      A     M      3.3;
      =     L      0.0;
      A(    ;
      A(    ;
      A     L      0.0;
      AN    M   2002.7;
      JNB   _001;
      L     0;
      T     MW  2150;
      SET   ;
      SAVE  ;
      CLR   ;
_001: A     BR;
      )     ;
      JNB   _002;
      L     0;
      T     MW  2152;
      SET   ;
      SAVE  ;
      CLR   ;
_002: A     BR;
      )     ;
      JNB   _003;
      L     0;
      T     MB  2154;
_003: NOP   0;
      A(    ;
      A(    ;
      A     L      0.0;
      AN    M   2002.5;
      JNB   _004;
      L     0;
      T     MW  2250;
      SET   ;
      SAVE  ;
      CLR   ;
_004: A     BR;
      )     ;
      JNB   _005;
      L     0;
      T     MW  2252;
      SET   ;
      SAVE  ;
      CLR   ;
_005: A     BR;
      )     ;
      JNB   _006;
      L     0;
      T     MB  2254;
_006: NOP   0;
NETWORK
TITLE =
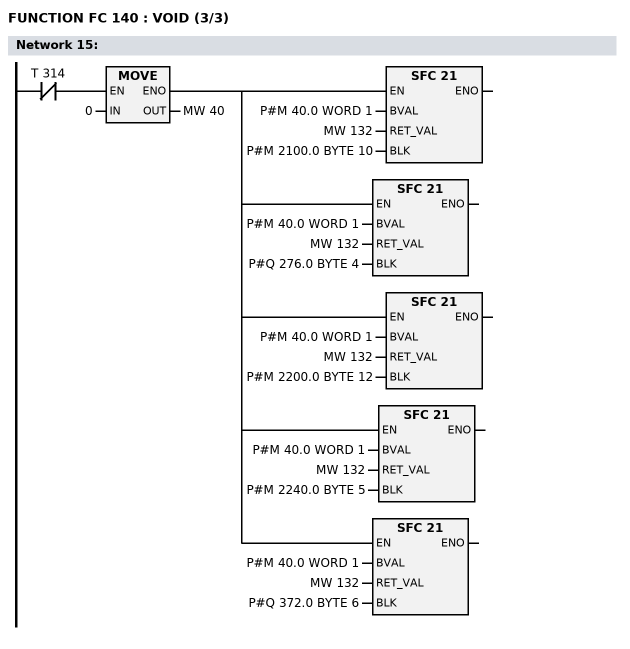

      AN    T    314;
      JNB   _007;
      L     0;
      T     MW    40;
      SET   ;
      SAVE  ;
      CLR   ;
_007: A     BR;
      =     L      0.0;
      A     L      0.0;
      JNB   _008;
      CALL SFC   21 (
           BVAL                     := P#M 40.0 WORD 1,
           RET_VAL                  := MW   132,
           BLK                      := P#M 2100.0 BYTE 10);
_008: NOP   0;
      A     L      0.0;
      JNB   _009;
      CALL SFC   21 (
           BVAL                     := P#M 40.0 WORD 1,
           RET_VAL                  := MW   132,
           BLK                      := P#Q 276.0 BYTE 4);
_009: NOP   0;
      A     L      0.0;
      JNB   _00a;
      CALL SFC   21 (
           BVAL                     := P#M 40.0 WORD 1,
           RET_VAL                  := MW   132,
           BLK                      := P#M 2200.0 BYTE 12);
_00a: NOP   0;
      A     L      0.0;
      JNB   _00b;
      CALL SFC   21 (
           BVAL                     := P#M 40.0 WORD 1,
           RET_VAL                  := MW   132,
           BLK                      := P#M 2240.0 BYTE 5);
_00b: NOP   0;
      A     L      0.0;
      JNB   _00c;
      CALL SFC   21 (
           BVAL                     := P#M 40.0 WORD 1,
           RET_VAL                  := MW   132,
           BLK                      := P#Q 372.0 BYTE 6);
_00c: NOP   0;
END_FUNCTION

FUNCTION_BLOCK FB 141
TITLE =
VERSION : 0.1


VAR
  S704_HOOK_PIN : FB 424;
  S704_DAECHA_LOCK : FB 424;
  S704_ELE : FB 424;
  S704_AIR_ELE : FB 424;
  S704_FF_OUT_CLAMP : FB 424;
END_VAR
BEGIN
NETWORK
TITLE =
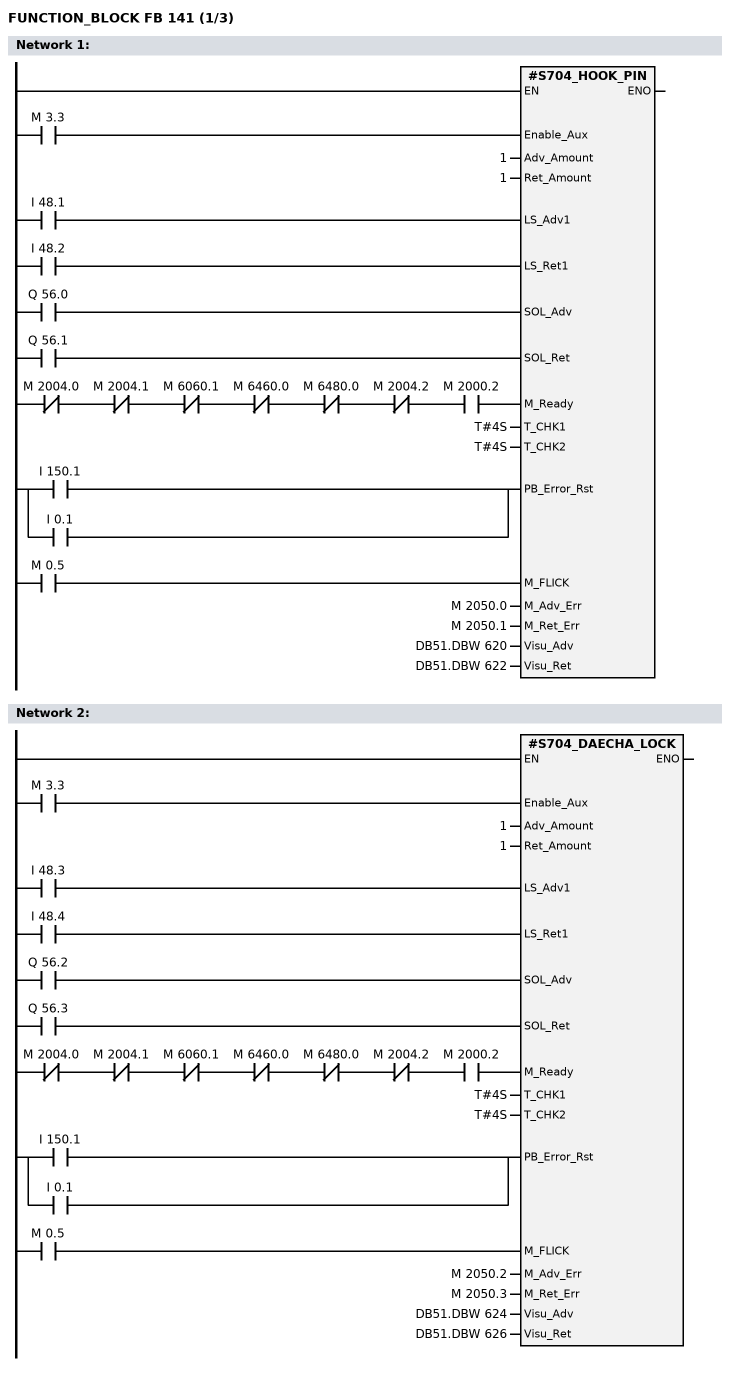

      A     M      3.3;
      =     L      0.0;
      BLD   103;
      A     I     48.1;
      =     L      0.1;
      BLD   103;
      A     I     48.2;
      =     L      0.2;
      BLD   103;
      A     Q     56.0;
      =     L      1.1;
      BLD   103;
      A     Q     56.1;
      =     L      1.2;
      BLD   103;
      AN    M   2004.0;
      AN    M   2004.1;
      AN    M   6060.1;
      AN    M   6460.0;
      AN    M   6480.0;
      AN    M   2004.2;
      A     M   2000.2;
      =     L      1.3;
      BLD   103;
      A(    ;
      O     I    150.1;
      O     I      0.1;
      )     ;
      =     L      1.5;
      BLD   103;
      A     M      0.5;
      =     L      1.6;
      BLD   103;
      CALL #S704_HOOK_PIN (
           Enable_Aux               := L      0.0,
           Adv_Amount               := 1,
           Ret_Amount               := 1,
           LS_Adv1                  := L      0.1,
           LS_Ret1                  := L      0.2,
           SOL_Adv                  := L      1.1,
           SOL_Ret                  := L      1.2,
           M_Ready                  := L      1.3,
           T_CHK1                   := T#4S,
           T_CHK2                   := T#4S,
           PB_Error_Rst             := L      1.5,
           M_FLICK                  := L      1.6,
           M_Adv_Err                := M   2050.0,
           M_Ret_Err                := M   2050.1,
           Visu_Adv                 := DB51.DBW  620,
           Visu_Ret                 := DB51.DBW  622);
      NOP   0;
NETWORK
TITLE =

      A     M      3.3;
      =     L      0.0;
      BLD   103;
      A     I     48.3;
      =     L      0.1;
      BLD   103;
      A     I     48.4;
      =     L      0.2;
      BLD   103;
      A     Q     56.2;
      =     L      1.1;
      BLD   103;
      A     Q     56.3;
      =     L      1.2;
      BLD   103;
      AN    M   2004.0;
      AN    M   2004.1;
      AN    M   6060.1;
      AN    M   6460.0;
      AN    M   6480.0;
      AN    M   2004.2;
      A     M   2000.2;
      =     L      1.3;
      BLD   103;
      A(    ;
      O     I    150.1;
      O     I      0.1;
      )     ;
      =     L      1.5;
      BLD   103;
      A     M      0.5;
      =     L      1.6;
      BLD   103;
      CALL #S704_DAECHA_LOCK (
           Enable_Aux               := L      0.0,
           Adv_Amount               := 1,
           Ret_Amount               := 1,
           LS_Adv1                  := L      0.1,
           LS_Ret1                  := L      0.2,
           SOL_Adv                  := L      1.1,
           SOL_Ret                  := L      1.2,
           M_Ready                  := L      1.3,
           T_CHK1                   := T#4S,
           T_CHK2                   := T#4S,
           PB_Error_Rst             := L      1.5,
           M_FLICK                  := L      1.6,
           M_Adv_Err                := M   2050.2,
           M_Ret_Err                := M   2050.3,
           Visu_Adv                 := DB51.DBW  624,
           Visu_Ret                 := DB51.DBW  626);
      NOP   0;
NETWORK
TITLE =
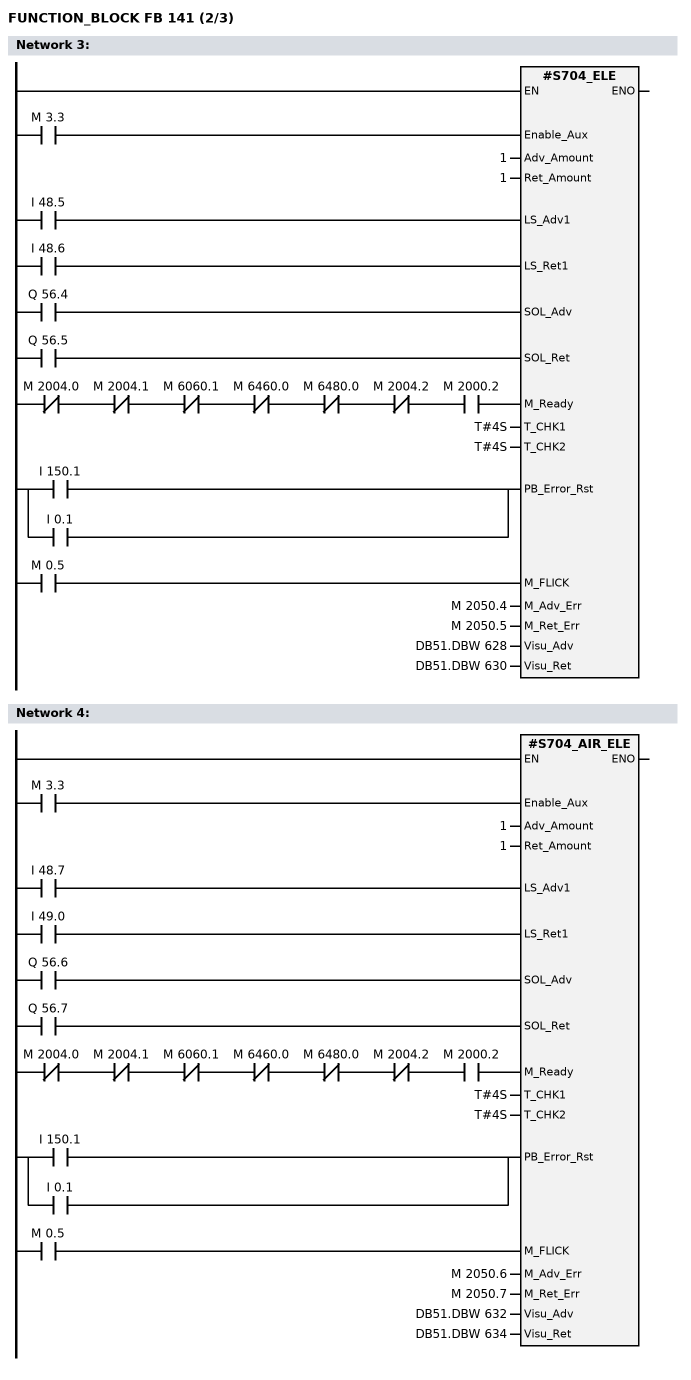

      A     M      3.3;
      =     L      0.0;
      BLD   103;
      A     I     48.5;
      =     L      0.1;
      BLD   103;
      A     I     48.6;
      =     L      0.2;
      BLD   103;
      A     Q     56.4;
      =     L      1.1;
      BLD   103;
      A     Q     56.5;
      =     L      1.2;
      BLD   103;
      AN    M   2004.0;
      AN    M   2004.1;
      AN    M   6060.1;
      AN    M   6460.0;
      AN    M   6480.0;
      AN    M   2004.2;
      A     M   2000.2;
      =     L      1.3;
      BLD   103;
      A(    ;
      O     I    150.1;
      O     I      0.1;
      )     ;
      =     L      1.5;
      BLD   103;
      A     M      0.5;
      =     L      1.6;
      BLD   103;
      CALL #S704_ELE (
           Enable_Aux               := L      0.0,
           Adv_Amount               := 1,
           Ret_Amount               := 1,
           LS_Adv1                  := L      0.1,
           LS_Ret1                  := L      0.2,
           SOL_Adv                  := L      1.1,
           SOL_Ret                  := L      1.2,
           M_Ready                  := L      1.3,
           T_CHK1                   := T#4S,
           T_CHK2                   := T#4S,
           PB_Error_Rst             := L      1.5,
           M_FLICK                  := L      1.6,
           M_Adv_Err                := M   2050.4,
           M_Ret_Err                := M   2050.5,
           Visu_Adv                 := DB51.DBW  628,
           Visu_Ret                 := DB51.DBW  630);
      NOP   0;
NETWORK
TITLE =

      A     M      3.3;
      =     L      0.0;
      BLD   103;
      A     I     48.7;
      =     L      0.1;
      BLD   103;
      A     I     49.0;
      =     L      0.2;
      BLD   103;
      A     Q     56.6;
      =     L      1.1;
      BLD   103;
      A     Q     56.7;
      =     L      1.2;
      BLD   103;
      AN    M   2004.0;
      AN    M   2004.1;
      AN    M   6060.1;
      AN    M   6460.0;
      AN    M   6480.0;
      AN    M   2004.2;
      A     M   2000.2;
      =     L      1.3;
      BLD   103;
      A(    ;
      O     I    150.1;
      O     I      0.1;
      )     ;
      =     L      1.5;
      BLD   103;
      A     M      0.5;
      =     L      1.6;
      BLD   103;
      CALL #S704_AIR_ELE (
           Enable_Aux               := L      0.0,
           Adv_Amount               := 1,
           Ret_Amount               := 1,
           LS_Adv1                  := L      0.1,
           LS_Ret1                  := L      0.2,
           SOL_Adv                  := L      1.1,
           SOL_Ret                  := L      1.2,
           M_Ready                  := L      1.3,
           T_CHK1                   := T#4S,
           T_CHK2                   := T#4S,
           PB_Error_Rst             := L      1.5,
           M_FLICK                  := L      1.6,
           M_Adv_Err                := M   2050.6,
           M_Ret_Err                := M   2050.7,
           Visu_Adv                 := DB51.DBW  632,
           Visu_Ret                 := DB51.DBW  634);
      NOP   0;
NETWORK
TITLE =
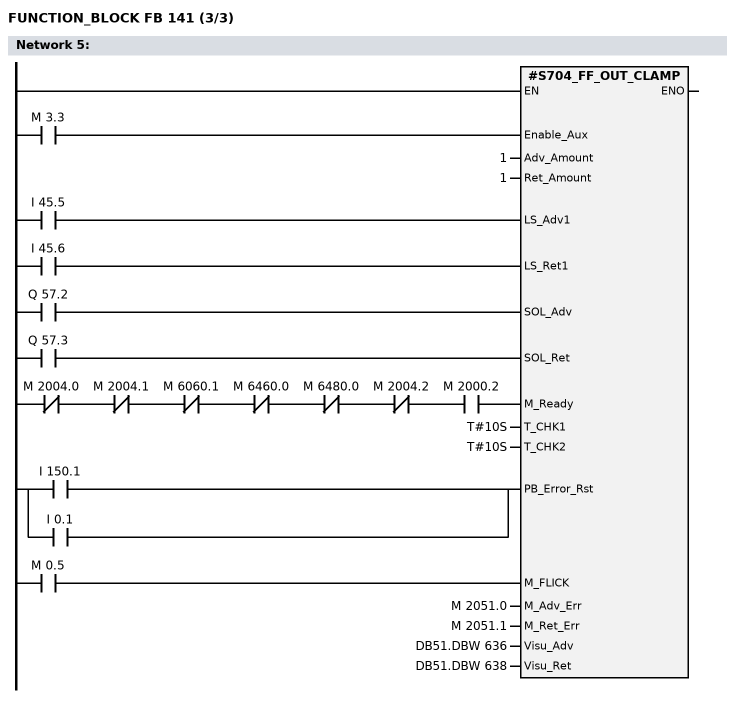

      A     M      3.3;
      =     L      0.0;
      BLD   103;
      A     I     45.5;
      =     L      0.1;
      BLD   103;
      A     I     45.6;
      =     L      0.2;
      BLD   103;
      A     Q     57.2;
      =     L      1.1;
      BLD   103;
      A     Q     57.3;
      =     L      1.2;
      BLD   103;
      AN    M   2004.0;
      AN    M   2004.1;
      AN    M   6060.1;
      AN    M   6460.0;
      AN    M   6480.0;
      AN    M   2004.2;
      A     M   2000.2;
      =     L      1.3;
      BLD   103;
      A(    ;
      O     I    150.1;
      O     I      0.1;
      )     ;
      =     L      1.5;
      BLD   103;
      A     M      0.5;
      =     L      1.6;
      BLD   103;
      CALL #S704_FF_OUT_CLAMP (
           Enable_Aux               := L      0.0,
           Adv_Amount               := 1,
           Ret_Amount               := 1,
           LS_Adv1                  := L      0.1,
           LS_Ret1                  := L      0.2,
           SOL_Adv                  := L      1.1,
           SOL_Ret                  := L      1.2,
           M_Ready                  := L      1.3,
           T_CHK1                   := T#10S,
           T_CHK2                   := T#10S,
           PB_Error_Rst             := L      1.5,
           M_FLICK                  := L      1.6,
           M_Adv_Err                := M   2051.0,
           M_Ret_Err                := M   2051.1,
           Visu_Adv                 := DB51.DBW  636,
           Visu_Ret                 := DB51.DBW  638);
      NOP   0;
END_FUNCTION_BLOCK

DATA_BLOCK DB 141
TITLE =
VERSION : 0.0

 FB 141
BEGIN
   S704_HOOK_PIN.Enable_Aux := FALSE;
   S704_HOOK_PIN.Adv_Amount := 0;
   S704_HOOK_PIN.Ret_Amount := 0;
   S704_HOOK_PIN.LS_Adv1 := FALSE;
   S704_HOOK_PIN.LS_Ret1 := FALSE;
   S704_HOOK_PIN.LS_Adv2 := FALSE;
   S704_HOOK_PIN.LS_Ret2 := FALSE;
   S704_HOOK_PIN.LS_Adv3 := FALSE;
   S704_HOOK_PIN.LS_Ret3 := FALSE;
   S704_HOOK_PIN.LS_Adv4 := FALSE;
   S704_HOOK_PIN.LS_Ret4 := FALSE;
   S704_HOOK_PIN.SOL_Adv := FALSE;
   S704_HOOK_PIN.SOL_Ret := FALSE;
   S704_HOOK_PIN.M_Ready := FALSE;
   S704_HOOK_PIN.T_CHK1 := T#0MS;
   S704_HOOK_PIN.T_CHK2 := T#0MS;
   S704_HOOK_PIN.PB_Lamp_CHK := FALSE;
   S704_HOOK_PIN.PB_Error_Rst := FALSE;
   S704_HOOK_PIN.M_FLICK := FALSE;
   S704_HOOK_PIN.M_Adv_Err := FALSE;
   S704_HOOK_PIN.M_Ret_Err := FALSE;
   S704_HOOK_PIN.LP_Adv := FALSE;
   S704_HOOK_PIN.LP_Ret := FALSE;
   S704_HOOK_PIN.Visu_Adv := W#16#0;
   S704_HOOK_PIN.Visu_Ret := W#16#0;
   S704_HOOK_PIN.Error_T1.IN := FALSE;
   S704_HOOK_PIN.Error_T1.PT := T#0MS;
   S704_HOOK_PIN.Error_T1.Q := FALSE;
   S704_HOOK_PIN.Error_T1.ET := T#0MS;
   S704_HOOK_PIN.Error_T1.STATE := B#16#0;
   S704_HOOK_PIN.Error_T1.STIME := T#0MS;
   S704_HOOK_PIN.Error_T1.ATIME := T#0MS;
   S704_HOOK_PIN.Error_T2.IN := FALSE;
   S704_HOOK_PIN.Error_T2.PT := T#0MS;
   S704_HOOK_PIN.Error_T2.Q := FALSE;
   S704_HOOK_PIN.Error_T2.ET := T#0MS;
   S704_HOOK_PIN.Error_T2.STATE := B#16#0;
   S704_HOOK_PIN.Error_T2.STIME := T#0MS;
   S704_HOOK_PIN.Error_T2.ATIME := T#0MS;
   S704_HOOK_PIN.CHK_Aux1 := FALSE;
   S704_HOOK_PIN.CHK_Aux2 := FALSE;
   S704_HOOK_PIN.Error_T1_DN := FALSE;
   S704_HOOK_PIN.Error_T2_DN := FALSE;
   S704_HOOK_PIN.Adv_Memo := FALSE;
   S704_HOOK_PIN.Visu_Adv_Arr[0] := FALSE;
   S704_HOOK_PIN.Visu_Adv_Arr[1] := FALSE;
   S704_HOOK_PIN.Visu_Adv_Arr[2] := FALSE;
   S704_HOOK_PIN.Visu_Adv_Arr[3] := FALSE;
   S704_HOOK_PIN.Visu_Adv_Arr[4] := FALSE;
   S704_HOOK_PIN.Visu_Adv_Arr[5] := FALSE;
   S704_HOOK_PIN.Visu_Adv_Arr[6] := FALSE;
   S704_HOOK_PIN.Visu_Adv_Arr[7] := FALSE;
   S704_HOOK_PIN.Visu_Adv_Arr[8] := FALSE;
   S704_HOOK_PIN.Visu_Adv_Arr[9] := FALSE;
   S704_HOOK_PIN.Visu_Adv_Arr[10] := FALSE;
   S704_HOOK_PIN.Visu_Adv_Arr[11] := FALSE;
   S704_HOOK_PIN.Visu_Adv_Arr[12] := FALSE;
   S704_HOOK_PIN.Visu_Adv_Arr[13] := FALSE;
   S704_HOOK_PIN.Visu_Adv_Arr[14] := FALSE;
   S704_HOOK_PIN.Visu_Adv_Arr[15] := FALSE;
   S704_HOOK_PIN.Visu_Ret_Arr[0] := FALSE;
   S704_HOOK_PIN.Visu_Ret_Arr[1] := FALSE;
   S704_HOOK_PIN.Visu_Ret_Arr[2] := FALSE;
   S704_HOOK_PIN.Visu_Ret_Arr[3] := FALSE;
   S704_HOOK_PIN.Visu_Ret_Arr[4] := FALSE;
   S704_HOOK_PIN.Visu_Ret_Arr[5] := FALSE;
   S704_HOOK_PIN.Visu_Ret_Arr[6] := FALSE;
   S704_HOOK_PIN.Visu_Ret_Arr[7] := FALSE;
   S704_HOOK_PIN.Visu_Ret_Arr[8] := FALSE;
   S704_HOOK_PIN.Visu_Ret_Arr[9] := FALSE;
   S704_HOOK_PIN.Visu_Ret_Arr[10] := FALSE;
   S704_HOOK_PIN.Visu_Ret_Arr[11] := FALSE;
   S704_HOOK_PIN.Visu_Ret_Arr[12] := FALSE;
   S704_HOOK_PIN.Visu_Ret_Arr[13] := FALSE;
   S704_HOOK_PIN.Visu_Ret_Arr[14] := FALSE;
   S704_HOOK_PIN.Visu_Ret_Arr[15] := FALSE;
   S704_HOOK_PIN.BLK_Move_Ret := 0;
   S704_HOOK_PIN.Enable := FALSE;
   S704_HOOK_PIN.Adv_End := FALSE;
   S704_HOOK_PIN.Ret_End := FALSE;
   S704_DAECHA_LOCK.Enable_Aux := FALSE;
   S704_DAECHA_LOCK.Adv_Amount := 0;
   S704_DAECHA_LOCK.Ret_Amount := 0;
   S704_DAECHA_LOCK.LS_Adv1 := FALSE;
   S704_DAECHA_LOCK.LS_Ret1 := FALSE;
   S704_DAECHA_LOCK.LS_Adv2 := FALSE;
   S704_DAECHA_LOCK.LS_Ret2 := FALSE;
   S704_DAECHA_LOCK.LS_Adv3 := FALSE;
   S704_DAECHA_LOCK.LS_Ret3 := FALSE;
   S704_DAECHA_LOCK.LS_Adv4 := FALSE;
   S704_DAECHA_LOCK.LS_Ret4 := FALSE;
   S704_DAECHA_LOCK.SOL_Adv := FALSE;
   S704_DAECHA_LOCK.SOL_Ret := FALSE;
   S704_DAECHA_LOCK.M_Ready := FALSE;
   S704_DAECHA_LOCK.T_CHK1 := T#0MS;
   S704_DAECHA_LOCK.T_CHK2 := T#0MS;
   S704_DAECHA_LOCK.PB_Lamp_CHK := FALSE;
   S704_DAECHA_LOCK.PB_Error_Rst := FALSE;
   S704_DAECHA_LOCK.M_FLICK := FALSE;
   S704_DAECHA_LOCK.M_Adv_Err := FALSE;
   S704_DAECHA_LOCK.M_Ret_Err := FALSE;
   S704_DAECHA_LOCK.LP_Adv := FALSE;
   S704_DAECHA_LOCK.LP_Ret := FALSE;
   S704_DAECHA_LOCK.Visu_Adv := W#16#0;
   S704_DAECHA_LOCK.Visu_Ret := W#16#0;
   S704_DAECHA_LOCK.Error_T1.IN := FALSE;
   S704_DAECHA_LOCK.Error_T1.PT := T#0MS;
   S704_DAECHA_LOCK.Error_T1.Q := FALSE;
   S704_DAECHA_LOCK.Error_T1.ET := T#0MS;
   S704_DAECHA_LOCK.Error_T1.STATE := B#16#0;
   S704_DAECHA_LOCK.Error_T1.STIME := T#0MS;
   S704_DAECHA_LOCK.Error_T1.ATIME := T#0MS;
   S704_DAECHA_LOCK.Error_T2.IN := FALSE;
   S704_DAECHA_LOCK.Error_T2.PT := T#0MS;
   S704_DAECHA_LOCK.Error_T2.Q := FALSE;
   S704_DAECHA_LOCK.Error_T2.ET := T#0MS;
   S704_DAECHA_LOCK.Error_T2.STATE := B#16#0;
   S704_DAECHA_LOCK.Error_T2.STIME := T#0MS;
   S704_DAECHA_LOCK.Error_T2.ATIME := T#0MS;
   S704_DAECHA_LOCK.CHK_Aux1 := FALSE;
   S704_DAECHA_LOCK.CHK_Aux2 := FALSE;
   S704_DAECHA_LOCK.Error_T1_DN := FALSE;
   S704_DAECHA_LOCK.Error_T2_DN := FALSE;
   S704_DAECHA_LOCK.Adv_Memo := FALSE;
   S704_DAECHA_LOCK.Visu_Adv_Arr[0] := FALSE;
   S704_DAECHA_LOCK.Visu_Adv_Arr[1] := FALSE;
   S704_DAECHA_LOCK.Visu_Adv_Arr[2] := FALSE;
   S704_DAECHA_LOCK.Visu_Adv_Arr[3] := FALSE;
   S704_DAECHA_LOCK.Visu_Adv_Arr[4] := FALSE;
   S704_DAECHA_LOCK.Visu_Adv_Arr[5] := FALSE;
   S704_DAECHA_LOCK.Visu_Adv_Arr[6] := FALSE;
   S704_DAECHA_LOCK.Visu_Adv_Arr[7] := FALSE;
   S704_DAECHA_LOCK.Visu_Adv_Arr[8] := FALSE;
   S704_DAECHA_LOCK.Visu_Adv_Arr[9] := FALSE;
   S704_DAECHA_LOCK.Visu_Adv_Arr[10] := FALSE;
   S704_DAECHA_LOCK.Visu_Adv_Arr[11] := FALSE;
   S704_DAECHA_LOCK.Visu_Adv_Arr[12] := FALSE;
   S704_DAECHA_LOCK.Visu_Adv_Arr[13] := FALSE;
   S704_DAECHA_LOCK.Visu_Adv_Arr[14] := FALSE;
   S704_DAECHA_LOCK.Visu_Adv_Arr[15] := FALSE;
   S704_DAECHA_LOCK.Visu_Ret_Arr[0] := FALSE;
   S704_DAECHA_LOCK.Visu_Ret_Arr[1] := FALSE;
   S704_DAECHA_LOCK.Visu_Ret_Arr[2] := FALSE;
   S704_DAECHA_LOCK.Visu_Ret_Arr[3] := FALSE;
   S704_DAECHA_LOCK.Visu_Ret_Arr[4] := FALSE;
   S704_DAECHA_LOCK.Visu_Ret_Arr[5] := FALSE;
   S704_DAECHA_LOCK.Visu_Ret_Arr[6] := FALSE;
   S704_DAECHA_LOCK.Visu_Ret_Arr[7] := FALSE;
   S704_DAECHA_LOCK.Visu_Ret_Arr[8] := FALSE;
   S704_DAECHA_LOCK.Visu_Ret_Arr[9] := FALSE;
   S704_DAECHA_LOCK.Visu_Ret_Arr[10] := FALSE;
   S704_DAECHA_LOCK.Visu_Ret_Arr[11] := FALSE;
   S704_DAECHA_LOCK.Visu_Ret_Arr[12] := FALSE;
   S704_DAECHA_LOCK.Visu_Ret_Arr[13] := FALSE;
   S704_DAECHA_LOCK.Visu_Ret_Arr[14] := FALSE;
   S704_DAECHA_LOCK.Visu_Ret_Arr[15] := FALSE;
   S704_DAECHA_LOCK.BLK_Move_Ret := 0;
   S704_DAECHA_LOCK.Enable := FALSE;
   S704_DAECHA_LOCK.Adv_End := FALSE;
   S704_DAECHA_LOCK.Ret_End := FALSE;
   S704_ELE.Enable_Aux := FALSE;
   S704_ELE.Adv_Amount := 0;
   S704_ELE.Ret_Amount := 0;
   S704_ELE.LS_Adv1 := FALSE;
   S704_ELE.LS_Ret1 := FALSE;
   S704_ELE.LS_Adv2 := FALSE;
   S704_ELE.LS_Ret2 := FALSE;
   S704_ELE.LS_Adv3 := FALSE;
   S704_ELE.LS_Ret3 := FALSE;
   S704_ELE.LS_Adv4 := FALSE;
   S704_ELE.LS_Ret4 := FALSE;
   S704_ELE.SOL_Adv := FALSE;
   S704_ELE.SOL_Ret := FALSE;
   S704_ELE.M_Ready := FALSE;
   S704_ELE.T_CHK1 := T#0MS;
   S704_ELE.T_CHK2 := T#0MS;
   S704_ELE.PB_Lamp_CHK := FALSE;
   S704_ELE.PB_Error_Rst := FALSE;
   S704_ELE.M_FLICK := FALSE;
   S704_ELE.M_Adv_Err := FALSE;
   S704_ELE.M_Ret_Err := FALSE;
   S704_ELE.LP_Adv := FALSE;
   S704_ELE.LP_Ret := FALSE;
   S704_ELE.Visu_Adv := W#16#0;
   S704_ELE.Visu_Ret := W#16#0;
   S704_ELE.Error_T1.IN := FALSE;
   S704_ELE.Error_T1.PT := T#0MS;
   S704_ELE.Error_T1.Q := FALSE;
   S704_ELE.Error_T1.ET := T#0MS;
   S704_ELE.Error_T1.STATE := B#16#0;
   S704_ELE.Error_T1.STIME := T#0MS;
   S704_ELE.Error_T1.ATIME := T#0MS;
   S704_ELE.Error_T2.IN := FALSE;
   S704_ELE.Error_T2.PT := T#0MS;
   S704_ELE.Error_T2.Q := FALSE;
   S704_ELE.Error_T2.ET := T#0MS;
   S704_ELE.Error_T2.STATE := B#16#0;
   S704_ELE.Error_T2.STIME := T#0MS;
   S704_ELE.Error_T2.ATIME := T#0MS;
   S704_ELE.CHK_Aux1 := FALSE;
   S704_ELE.CHK_Aux2 := FALSE;
   S704_ELE.Error_T1_DN := FALSE;
   S704_ELE.Error_T2_DN := FALSE;
   S704_ELE.Adv_Memo := FALSE;
   S704_ELE.Visu_Adv_Arr[0] := FALSE;
   S704_ELE.Visu_Adv_Arr[1] := FALSE;
   S704_ELE.Visu_Adv_Arr[2] := FALSE;
   S704_ELE.Visu_Adv_Arr[3] := FALSE;
   S704_ELE.Visu_Adv_Arr[4] := FALSE;
   S704_ELE.Visu_Adv_Arr[5] := FALSE;
   S704_ELE.Visu_Adv_Arr[6] := FALSE;
   S704_ELE.Visu_Adv_Arr[7] := FALSE;
   S704_ELE.Visu_Adv_Arr[8] := FALSE;
   S704_ELE.Visu_Adv_Arr[9] := FALSE;
   S704_ELE.Visu_Adv_Arr[10] := FALSE;
   S704_ELE.Visu_Adv_Arr[11] := FALSE;
   S704_ELE.Visu_Adv_Arr[12] := FALSE;
   S704_ELE.Visu_Adv_Arr[13] := FALSE;
   S704_ELE.Visu_Adv_Arr[14] := FALSE;
   S704_ELE.Visu_Adv_Arr[15] := FALSE;
   S704_ELE.Visu_Ret_Arr[0] := FALSE;
   S704_ELE.Visu_Ret_Arr[1] := FALSE;
   S704_ELE.Visu_Ret_Arr[2] := FALSE;
   S704_ELE.Visu_Ret_Arr[3] := FALSE;
   S704_ELE.Visu_Ret_Arr[4] := FALSE;
   S704_ELE.Visu_Ret_Arr[5] := FALSE;
   S704_ELE.Visu_Ret_Arr[6] := FALSE;
   S704_ELE.Visu_Ret_Arr[7] := FALSE;
   S704_ELE.Visu_Ret_Arr[8] := FALSE;
   S704_ELE.Visu_Ret_Arr[9] := FALSE;
   S704_ELE.Visu_Ret_Arr[10] := FALSE;
   S704_ELE.Visu_Ret_Arr[11] := FALSE;
   S704_ELE.Visu_Ret_Arr[12] := FALSE;
   S704_ELE.Visu_Ret_Arr[13] := FALSE;
   S704_ELE.Visu_Ret_Arr[14] := FALSE;
   S704_ELE.Visu_Ret_Arr[15] := FALSE;
   S704_ELE.BLK_Move_Ret := 0;
   S704_ELE.Enable := FALSE;
   S704_ELE.Adv_End := FALSE;
   S704_ELE.Ret_End := FALSE;
   S704_AIR_ELE.Enable_Aux := FALSE;
   S704_AIR_ELE.Adv_Amount := 0;
   S704_AIR_ELE.Ret_Amount := 0;
   S704_AIR_ELE.LS_Adv1 := FALSE;
   S704_AIR_ELE.LS_Ret1 := FALSE;
   S704_AIR_ELE.LS_Adv2 := FALSE;
   S704_AIR_ELE.LS_Ret2 := FALSE;
   S704_AIR_ELE.LS_Adv3 := FALSE;
   S704_AIR_ELE.LS_Ret3 := FALSE;
   S704_AIR_ELE.LS_Adv4 := FALSE;
   S704_AIR_ELE.LS_Ret4 := FALSE;
   S704_AIR_ELE.SOL_Adv := FALSE;
   S704_AIR_ELE.SOL_Ret := FALSE;
   S704_AIR_ELE.M_Ready := FALSE;
   S704_AIR_ELE.T_CHK1 := T#0MS;
   S704_AIR_ELE.T_CHK2 := T#0MS;
   S704_AIR_ELE.PB_Lamp_CHK := FALSE;
   S704_AIR_ELE.PB_Error_Rst := FALSE;
   S704_AIR_ELE.M_FLICK := FALSE;
   S704_AIR_ELE.M_Adv_Err := FALSE;
   S704_AIR_ELE.M_Ret_Err := FALSE;
   S704_AIR_ELE.LP_Adv := FALSE;
   S704_AIR_ELE.LP_Ret := FALSE;
   S704_AIR_ELE.Visu_Adv := W#16#0;
   S704_AIR_ELE.Visu_Ret := W#16#0;
   S704_AIR_ELE.Error_T1.IN := FALSE;
   S704_AIR_ELE.Error_T1.PT := T#0MS;
   S704_AIR_ELE.Error_T1.Q := FALSE;
   S704_AIR_ELE.Error_T1.ET := T#0MS;
   S704_AIR_ELE.Error_T1.STATE := B#16#0;
   S704_AIR_ELE.Error_T1.STIME := T#0MS;
   S704_AIR_ELE.Error_T1.ATIME := T#0MS;
   S704_AIR_ELE.Error_T2.IN := FALSE;
   S704_AIR_ELE.Error_T2.PT := T#0MS;
   S704_AIR_ELE.Error_T2.Q := FALSE;
   S704_AIR_ELE.Error_T2.ET := T#0MS;
   S704_AIR_ELE.Error_T2.STATE := B#16#0;
   S704_AIR_ELE.Error_T2.STIME := T#0MS;
   S704_AIR_ELE.Error_T2.ATIME := T#0MS;
   S704_AIR_ELE.CHK_Aux1 := FALSE;
   S704_AIR_ELE.CHK_Aux2 := FALSE;
   S704_AIR_ELE.Error_T1_DN := FALSE;
   S704_AIR_ELE.Error_T2_DN := FALSE;
   S704_AIR_ELE.Adv_Memo := FALSE;
   S704_AIR_ELE.Visu_Adv_Arr[0] := FALSE;
   S704_AIR_ELE.Visu_Adv_Arr[1] := FALSE;
   S704_AIR_ELE.Visu_Adv_Arr[2] := FALSE;
   S704_AIR_ELE.Visu_Adv_Arr[3] := FALSE;
   S704_AIR_ELE.Visu_Adv_Arr[4] := FALSE;
   S704_AIR_ELE.Visu_Adv_Arr[5] := FALSE;
   S704_AIR_ELE.Visu_Adv_Arr[6] := FALSE;
   S704_AIR_ELE.Visu_Adv_Arr[7] := FALSE;
   S704_AIR_ELE.Visu_Adv_Arr[8] := FALSE;
   S704_AIR_ELE.Visu_Adv_Arr[9] := FALSE;
   S704_AIR_ELE.Visu_Adv_Arr[10] := FALSE;
   S704_AIR_ELE.Visu_Adv_Arr[11] := FALSE;
   S704_AIR_ELE.Visu_Adv_Arr[12] := FALSE;
   S704_AIR_ELE.Visu_Adv_Arr[13] := FALSE;
   S704_AIR_ELE.Visu_Adv_Arr[14] := FALSE;
   S704_AIR_ELE.Visu_Adv_Arr[15] := FALSE;
   S704_AIR_ELE.Visu_Ret_Arr[0] := FALSE;
   S704_AIR_ELE.Visu_Ret_Arr[1] := FALSE;
   S704_AIR_ELE.Visu_Ret_Arr[2] := FALSE;
   S704_AIR_ELE.Visu_Ret_Arr[3] := FALSE;
   S704_AIR_ELE.Visu_Ret_Arr[4] := FALSE;
   S704_AIR_ELE.Visu_Ret_Arr[5] := FALSE;
   S704_AIR_ELE.Visu_Ret_Arr[6] := FALSE;
   S704_AIR_ELE.Visu_Ret_Arr[7] := FALSE;
   S704_AIR_ELE.Visu_Ret_Arr[8] := FALSE;
   S704_AIR_ELE.Visu_Ret_Arr[9] := FALSE;
   S704_AIR_ELE.Visu_Ret_Arr[10] := FALSE;
   S704_AIR_ELE.Visu_Ret_Arr[11] := FALSE;
   S704_AIR_ELE.Visu_Ret_Arr[12] := FALSE;
   S704_AIR_ELE.Visu_Ret_Arr[13] := FALSE;
   S704_AIR_ELE.Visu_Ret_Arr[14] := FALSE;
   S704_AIR_ELE.Visu_Ret_Arr[15] := FALSE;
   S704_AIR_ELE.BLK_Move_Ret := 0;
   S704_AIR_ELE.Enable := FALSE;
   S704_AIR_ELE.Adv_End := FALSE;
   S704_AIR_ELE.Ret_End := FALSE;
   S704_FF_OUT_CLAMP.Enable_Aux := FALSE;
   S704_FF_OUT_CLAMP.Adv_Amount := 0;
   S704_FF_OUT_CLAMP.Ret_Amount := 0;
   S704_FF_OUT_CLAMP.LS_Adv1 := FALSE;
   S704_FF_OUT_CLAMP.LS_Ret1 := FALSE;
   S704_FF_OUT_CLAMP.LS_Adv2 := FALSE;
   S704_FF_OUT_CLAMP.LS_Ret2 := FALSE;
   S704_FF_OUT_CLAMP.LS_Adv3 := FALSE;
   S704_FF_OUT_CLAMP.LS_Ret3 := FALSE;
   S704_FF_OUT_CLAMP.LS_Adv4 := FALSE;
   S704_FF_OUT_CLAMP.LS_Ret4 := FALSE;
   S704_FF_OUT_CLAMP.SOL_Adv := FALSE;
   S704_FF_OUT_CLAMP.SOL_Ret := FALSE;
   S704_FF_OUT_CLAMP.M_Ready := FALSE;
   S704_FF_OUT_CLAMP.T_CHK1 := T#0MS;
   S704_FF_OUT_CLAMP.T_CHK2 := T#0MS;
   S704_FF_OUT_CLAMP.PB_Lamp_CHK := FALSE;
   S704_FF_OUT_CLAMP.PB_Error_Rst := FALSE;
   S704_FF_OUT_CLAMP.M_FLICK := FALSE;
   S704_FF_OUT_CLAMP.M_Adv_Err := FALSE;
   S704_FF_OUT_CLAMP.M_Ret_Err := FALSE;
   S704_FF_OUT_CLAMP.LP_Adv := FALSE;
   S704_FF_OUT_CLAMP.LP_Ret := FALSE;
   S704_FF_OUT_CLAMP.Visu_Adv := W#16#0;
   S704_FF_OUT_CLAMP.Visu_Ret := W#16#0;
   S704_FF_OUT_CLAMP.Error_T1.IN := FALSE;
   S704_FF_OUT_CLAMP.Error_T1.PT := T#0MS;
   S704_FF_OUT_CLAMP.Error_T1.Q := FALSE;
   S704_FF_OUT_CLAMP.Error_T1.ET := T#0MS;
   S704_FF_OUT_CLAMP.Error_T1.STATE := B#16#0;
   S704_FF_OUT_CLAMP.Error_T1.STIME := T#0MS;
   S704_FF_OUT_CLAMP.Error_T1.ATIME := T#0MS;
   S704_FF_OUT_CLAMP.Error_T2.IN := FALSE;
   S704_FF_OUT_CLAMP.Error_T2.PT := T#0MS;
   S704_FF_OUT_CLAMP.Error_T2.Q := FALSE;
   S704_FF_OUT_CLAMP.Error_T2.ET := T#0MS;
   S704_FF_OUT_CLAMP.Error_T2.STATE := B#16#0;
   S704_FF_OUT_CLAMP.Error_T2.STIME := T#0MS;
   S704_FF_OUT_CLAMP.Error_T2.ATIME := T#0MS;
   S704_FF_OUT_CLAMP.CHK_Aux1 := FALSE;
   S704_FF_OUT_CLAMP.CHK_Aux2 := FALSE;
   S704_FF_OUT_CLAMP.Error_T1_DN := FALSE;
   S704_FF_OUT_CLAMP.Error_T2_DN := FALSE;
   S704_FF_OUT_CLAMP.Adv_Memo := FALSE;
   S704_FF_OUT_CLAMP.Visu_Adv_Arr[0] := FALSE;
   S704_FF_OUT_CLAMP.Visu_Adv_Arr[1] := FALSE;
   S704_FF_OUT_CLAMP.Visu_Adv_Arr[2] := FALSE;
   S704_FF_OUT_CLAMP.Visu_Adv_Arr[3] := FALSE;
   S704_FF_OUT_CLAMP.Visu_Adv_Arr[4] := FALSE;
   S704_FF_OUT_CLAMP.Visu_Adv_Arr[5] := FALSE;
   S704_FF_OUT_CLAMP.Visu_Adv_Arr[6] := FALSE;
   S704_FF_OUT_CLAMP.Visu_Adv_Arr[7] := FALSE;
   S704_FF_OUT_CLAMP.Visu_Adv_Arr[8] := FALSE;
   S704_FF_OUT_CLAMP.Visu_Adv_Arr[9] := FALSE;
   S704_FF_OUT_CLAMP.Visu_Adv_Arr[10] := FALSE;
   S704_FF_OUT_CLAMP.Visu_Adv_Arr[11] := FALSE;
   S704_FF_OUT_CLAMP.Visu_Adv_Arr[12] := FALSE;
   S704_FF_OUT_CLAMP.Visu_Adv_Arr[13] := FALSE;
   S704_FF_OUT_CLAMP.Visu_Adv_Arr[14] := FALSE;
   S704_FF_OUT_CLAMP.Visu_Adv_Arr[15] := FALSE;
   S704_FF_OUT_CLAMP.Visu_Ret_Arr[0] := FALSE;
   S704_FF_OUT_CLAMP.Visu_Ret_Arr[1] := FALSE;
   S704_FF_OUT_CLAMP.Visu_Ret_Arr[2] := FALSE;
   S704_FF_OUT_CLAMP.Visu_Ret_Arr[3] := FALSE;
   S704_FF_OUT_CLAMP.Visu_Ret_Arr[4] := FALSE;
   S704_FF_OUT_CLAMP.Visu_Ret_Arr[5] := FALSE;
   S704_FF_OUT_CLAMP.Visu_Ret_Arr[6] := FALSE;
   S704_FF_OUT_CLAMP.Visu_Ret_Arr[7] := FALSE;
   S704_FF_OUT_CLAMP.Visu_Ret_Arr[8] := FALSE;
   S704_FF_OUT_CLAMP.Visu_Ret_Arr[9] := FALSE;
   S704_FF_OUT_CLAMP.Visu_Ret_Arr[10] := FALSE;
   S704_FF_OUT_CLAMP.Visu_Ret_Arr[11] := FALSE;
   S704_FF_OUT_CLAMP.Visu_Ret_Arr[12] := FALSE;
   S704_FF_OUT_CLAMP.Visu_Ret_Arr[13] := FALSE;
   S704_FF_OUT_CLAMP.Visu_Ret_Arr[14] := FALSE;
   S704_FF_OUT_CLAMP.Visu_Ret_Arr[15] := FALSE;
   S704_FF_OUT_CLAMP.BLK_Move_Ret := 0;
   S704_FF_OUT_CLAMP.Enable := FALSE;
   S704_FF_OUT_CLAMP.Adv_End := FALSE;
   S704_FF_OUT_CLAMP.Ret_End := FALSE;
END_DATA_BLOCK

FUNCTION FC 141 : VOID
TITLE =
VERSION : 0.1

BEGIN
NETWORK
TITLE =
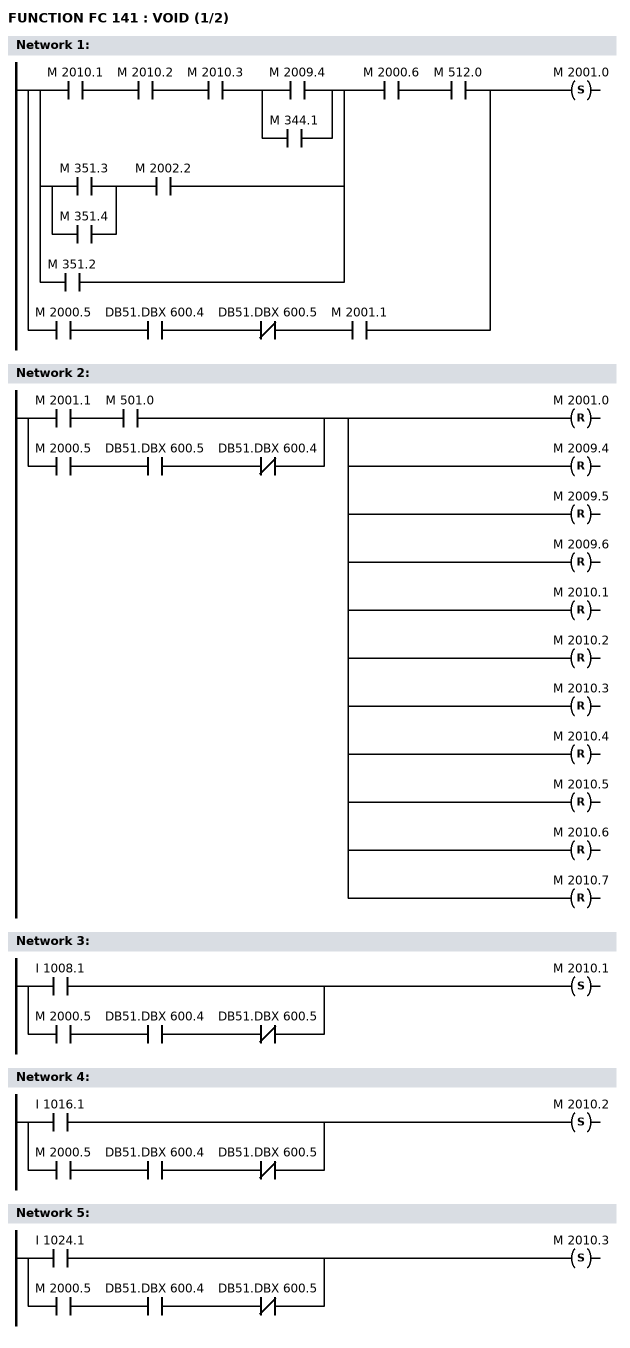

      A(    ;
      A     M   2010.1;
      A     M   2010.2;
      A     M   2010.3;
      A(    ;
      O     M   2009.4;
      O     M    344.1;
      )     ;
      O     ;
      A(    ;
      O     M    351.3;
      O     M    351.4;
      )     ;
      A     M   2002.2;
      O     M    351.2;
      )     ;
      A     M   2000.6;
      A     M    512.0;
      O     ;
      A     M   2000.5;
      A     DB51.DBX  600.4;
      AN    DB51.DBX  600.5;
      A     M   2001.1;
      S     M   2001.0;
NETWORK
TITLE =

      A     M   2001.1;
      A     M    501.0;
      O     ;
      A     M   2000.5;
      A     DB51.DBX  600.5;
      AN    DB51.DBX  600.4;
      R     M   2001.0;
      R     M   2009.4;
      R     M   2009.5;
      R     M   2009.6;
      R     M   2010.1;
      R     M   2010.2;
      R     M   2010.3;
      R     M   2010.4;
      R     M   2010.5;
      R     M   2010.6;
      R     M   2010.7;
NETWORK
TITLE =

      O     I   1008.1;
      O     ;
      A     M   2000.5;
      A     DB51.DBX  600.4;
      AN    DB51.DBX  600.5;
      S     M   2010.1;
NETWORK
TITLE =

      O     I   1016.1;
      O     ;
      A     M   2000.5;
      A     DB51.DBX  600.4;
      AN    DB51.DBX  600.5;
      S     M   2010.2;
NETWORK
TITLE =

      O     I   1024.1;
      O     ;
      A     M   2000.5;
      A     DB51.DBX  600.4;
      AN    DB51.DBX  600.5;
      S     M   2010.3;
NETWORK
TITLE =
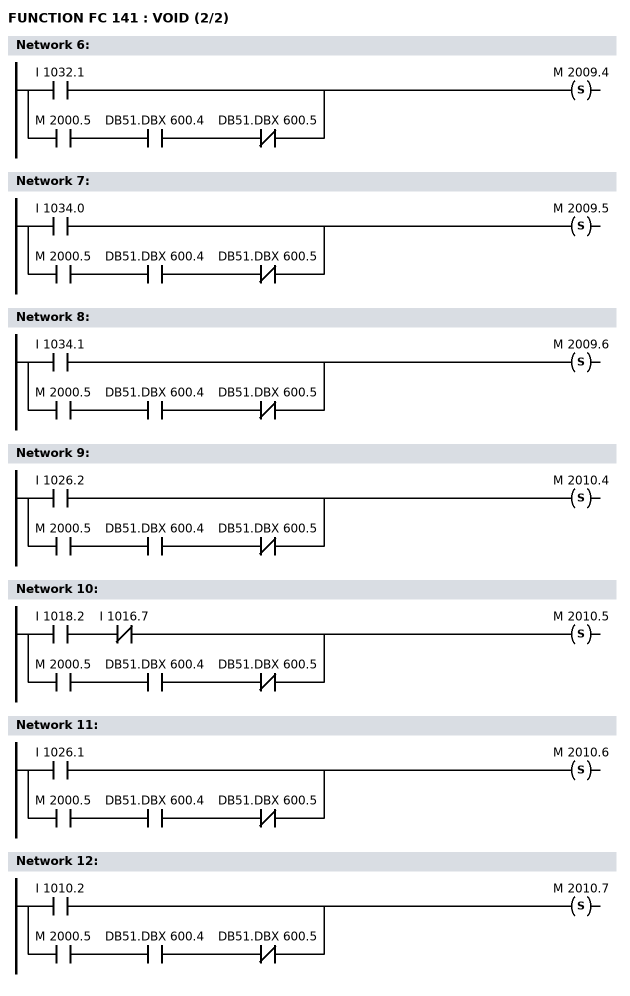

      O     I   1032.1;
      O     ;
      A     M   2000.5;
      A     DB51.DBX  600.4;
      AN    DB51.DBX  600.5;
      S     M   2009.4;
NETWORK
TITLE =

      O     I   1034.0;
      O     ;
      A     M   2000.5;
      A     DB51.DBX  600.4;
      AN    DB51.DBX  600.5;
      S     M   2009.5;
NETWORK
TITLE =

      O     I   1034.1;
      O     ;
      A     M   2000.5;
      A     DB51.DBX  600.4;
      AN    DB51.DBX  600.5;
      S     M   2009.6;
NETWORK
TITLE =

      O     I   1026.2;
      O     ;
      A     M   2000.5;
      A     DB51.DBX  600.4;
      AN    DB51.DBX  600.5;
      S     M   2010.4;
NETWORK
TITLE =

      A     I   1018.2;
      AN    I   1016.7;
      O     ;
      A     M   2000.5;
      A     DB51.DBX  600.4;
      AN    DB51.DBX  600.5;
      S     M   2010.5;
NETWORK
TITLE =

      O     I   1026.1;
      O     ;
      A     M   2000.5;
      A     DB51.DBX  600.4;
      AN    DB51.DBX  600.5;
      S     M   2010.6;
NETWORK
TITLE =

      O     I   1010.2;
      O     ;
      A     M   2000.5;
      A     DB51.DBX  600.4;
      AN    DB51.DBX  600.5;
      S     M   2010.7;
END_FUNCTION

FUNCTION_BLOCK FB 142
TITLE =
VERSION : 0.1

BEGIN
NETWORK
TITLE =
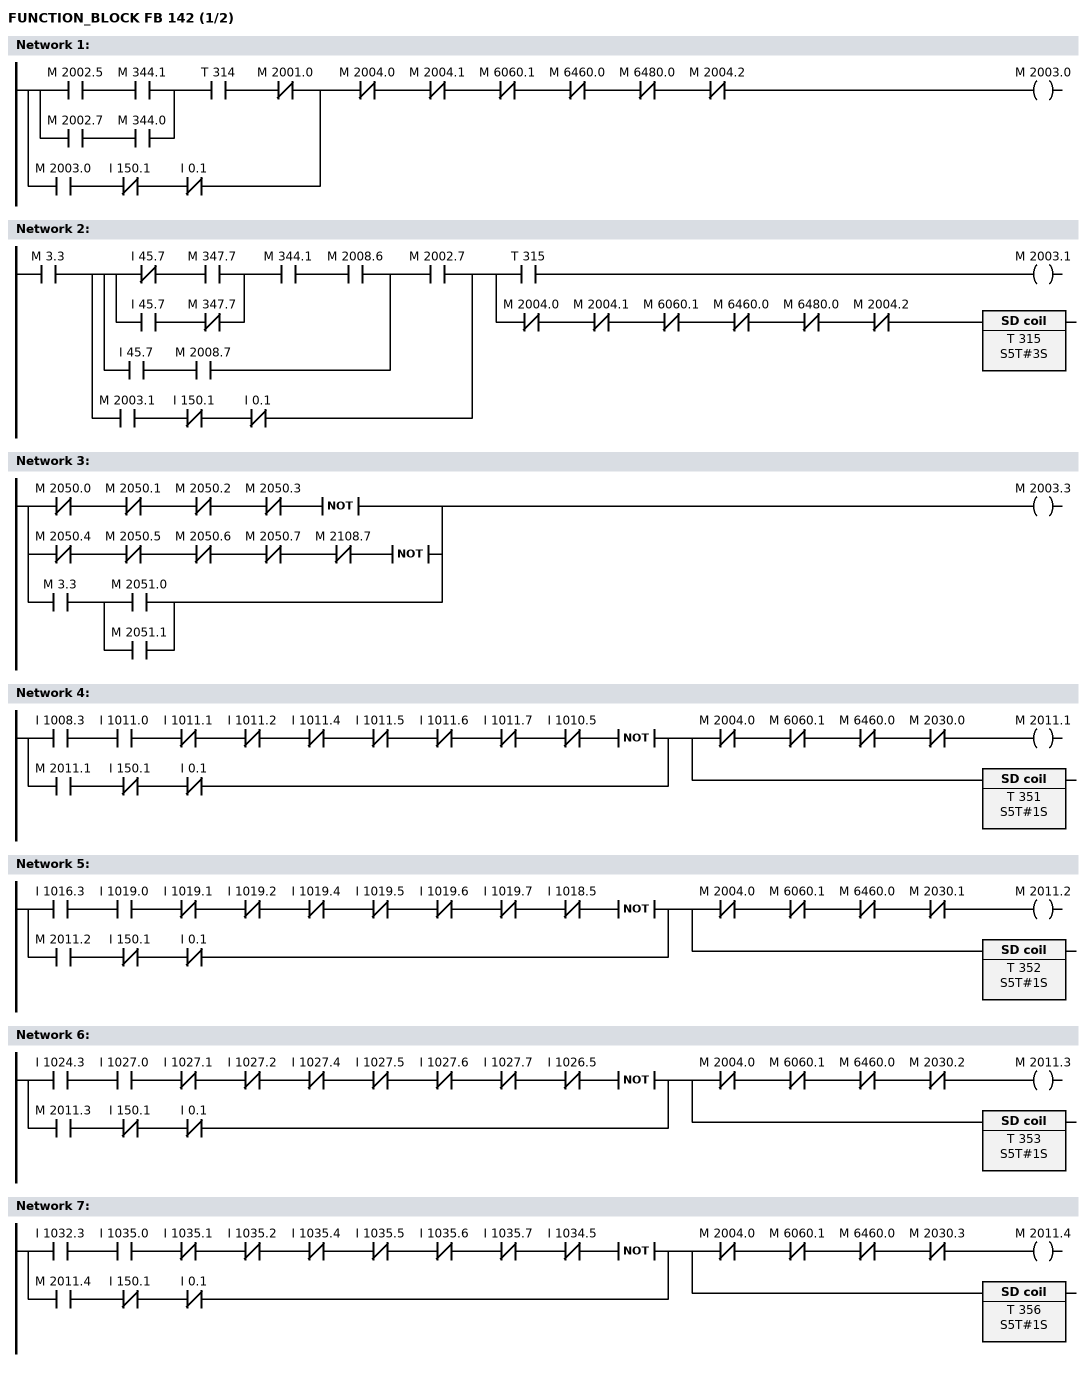

      A(    ;
      A(    ;
      A     M   2002.5;
      A     M    344.1;
      O     ;
      A     M   2002.7;
      A     M    344.0;
      )     ;
      A     T    314;
      AN    M   2001.0;
      O     ;
      A     M   2003.0;
      AN    I    150.1;
      AN    I      0.1;
      )     ;
      AN    M   2004.0;
      AN    M   2004.1;
      AN    M   6060.1;
      AN    M   6460.0;
      AN    M   6480.0;
      AN    M   2004.2;
      =     M   2003.0;
NETWORK
TITLE =

      A     M      3.3;
      A(    ;
      A(    ;
      A(    ;
      AN    I     45.7;
      A     M    347.7;
      O     ;
      A     I     45.7;
      AN    M    347.7;
      )     ;
      A     M    344.1;
      A     M   2008.6;
      O     ;
      A     I     45.7;
      A     M   2008.7;
      )     ;
      A     M   2002.7;
      O     ;
      A     M   2003.1;
      AN    I    150.1;
      AN    I      0.1;
      )     ;
      =     L      0.0;
      A     L      0.0;
      A     T    315;
      =     M   2003.1;
      A     L      0.0;
      AN    M   2004.0;
      AN    M   2004.1;
      AN    M   6060.1;
      AN    M   6460.0;
      AN    M   6480.0;
      AN    M   2004.2;
      L     S5T#3S;
      SD    T    315;
NETWORK
TITLE =

      AN    M   2050.0;
      AN    M   2050.1;
      AN    M   2050.2;
      AN    M   2050.3;
      NOT   ;
      O(    ;
      AN    M   2050.4;
      AN    M   2050.5;
      AN    M   2050.6;
      AN    M   2050.7;
      AN    M   2108.7;
      NOT   ;
      )     ;
      O     ;
      A     M      3.3;
      A(    ;
      O     M   2051.0;
      O     M   2051.1;
      )     ;
      =     M   2003.3;
NETWORK
TITLE =

      A     I   1008.3;
      A     I   1011.0;
      AN    I   1011.1;
      AN    I   1011.2;
      AN    I   1011.4;
      AN    I   1011.5;
      AN    I   1011.6;
      AN    I   1011.7;
      AN    I   1010.5;
      NOT   ;
      O     ;
      A     M   2011.1;
      AN    I    150.1;
      AN    I      0.1;
      =     L      0.0;
      A     L      0.0;
      AN    M   2004.0;
      AN    M   6060.1;
      AN    M   6460.0;
      AN    M   2030.0;
      =     M   2011.1;
      A     L      0.0;
      BLD   102;
      L     S5T#1S;
      SD    T    351;
NETWORK
TITLE =

      A     I   1016.3;
      A     I   1019.0;
      AN    I   1019.1;
      AN    I   1019.2;
      AN    I   1019.4;
      AN    I   1019.5;
      AN    I   1019.6;
      AN    I   1019.7;
      AN    I   1018.5;
      NOT   ;
      O     ;
      A     M   2011.2;
      AN    I    150.1;
      AN    I      0.1;
      =     L      0.0;
      A     L      0.0;
      AN    M   2004.0;
      AN    M   6060.1;
      AN    M   6460.0;
      AN    M   2030.1;
      =     M   2011.2;
      A     L      0.0;
      BLD   102;
      L     S5T#1S;
      SD    T    352;
NETWORK
TITLE =

      A     I   1024.3;
      A     I   1027.0;
      AN    I   1027.1;
      AN    I   1027.2;
      AN    I   1027.4;
      AN    I   1027.5;
      AN    I   1027.6;
      AN    I   1027.7;
      AN    I   1026.5;
      NOT   ;
      O     ;
      A     M   2011.3;
      AN    I    150.1;
      AN    I      0.1;
      =     L      0.0;
      A     L      0.0;
      AN    M   2004.0;
      AN    M   6060.1;
      AN    M   6460.0;
      AN    M   2030.2;
      =     M   2011.3;
      A     L      0.0;
      BLD   102;
      L     S5T#1S;
      SD    T    353;
NETWORK
TITLE =

      A     I   1032.3;
      A     I   1035.0;
      AN    I   1035.1;
      AN    I   1035.2;
      AN    I   1035.4;
      AN    I   1035.5;
      AN    I   1035.6;
      AN    I   1035.7;
      AN    I   1034.5;
      NOT   ;
      O     ;
      A     M   2011.4;
      AN    I    150.1;
      AN    I      0.1;
      =     L      0.0;
      A     L      0.0;
      AN    M   2004.0;
      AN    M   6060.1;
      AN    M   6460.0;
      AN    M   2030.3;
      =     M   2011.4;
      A     L      0.0;
      BLD   102;
      L     S5T#1S;
      SD    T    356;
NETWORK
TITLE =
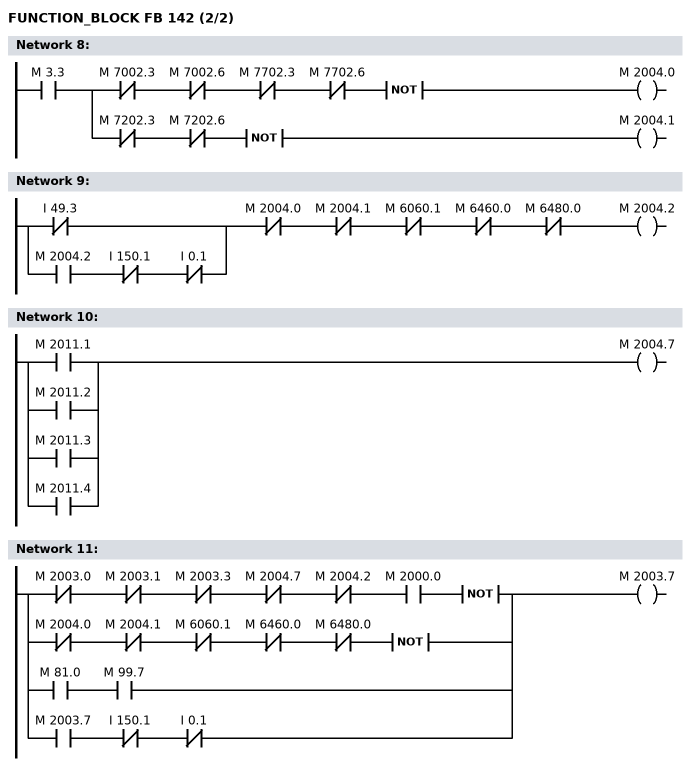

      A     M      3.3;
      =     L      0.0;
      A     L      0.0;
      AN    M   7002.3;
      AN    M   7002.6;
      AN    M   7702.3;
      AN    M   7702.6;
      NOT   ;
      =     M   2004.0;
      A     L      0.0;
      AN    M   7202.3;
      AN    M   7202.6;
      NOT   ;
      =     M   2004.1;
NETWORK
TITLE =

      A(    ;
      ON    I     49.3;
      O     ;
      A     M   2004.2;
      AN    I    150.1;
      AN    I      0.1;
      )     ;
      AN    M   2004.0;
      AN    M   2004.1;
      AN    M   6060.1;
      AN    M   6460.0;
      AN    M   6480.0;
      =     M   2004.2;
NETWORK
TITLE =

      O     M   2011.1;
      O     M   2011.2;
      O     M   2011.3;
      O     M   2011.4;
      =     M   2004.7;
NETWORK
TITLE =

      AN    M   2003.0;
      AN    M   2003.1;
      AN    M   2003.3;
      AN    M   2004.7;
      AN    M   2004.2;
      A     M   2000.0;
      NOT   ;
      O(    ;
      AN    M   2004.0;
      AN    M   2004.1;
      AN    M   6060.1;
      AN    M   6460.0;
      AN    M   6480.0;
      NOT   ;
      )     ;
      O     ;
      A     M     81.0;
      A     M     99.7;
      O     ;
      A     M   2003.7;
      AN    I    150.1;
      AN    I      0.1;
      =     M   2003.7;
END_FUNCTION_BLOCK

DATA_BLOCK DB 142
TITLE =
VERSION : 0.0

 FB 142
BEGIN
END_DATA_BLOCK

FUNCTION FC 142 : VOID
TITLE =
VERSION : 0.1

BEGIN
NETWORK
TITLE =
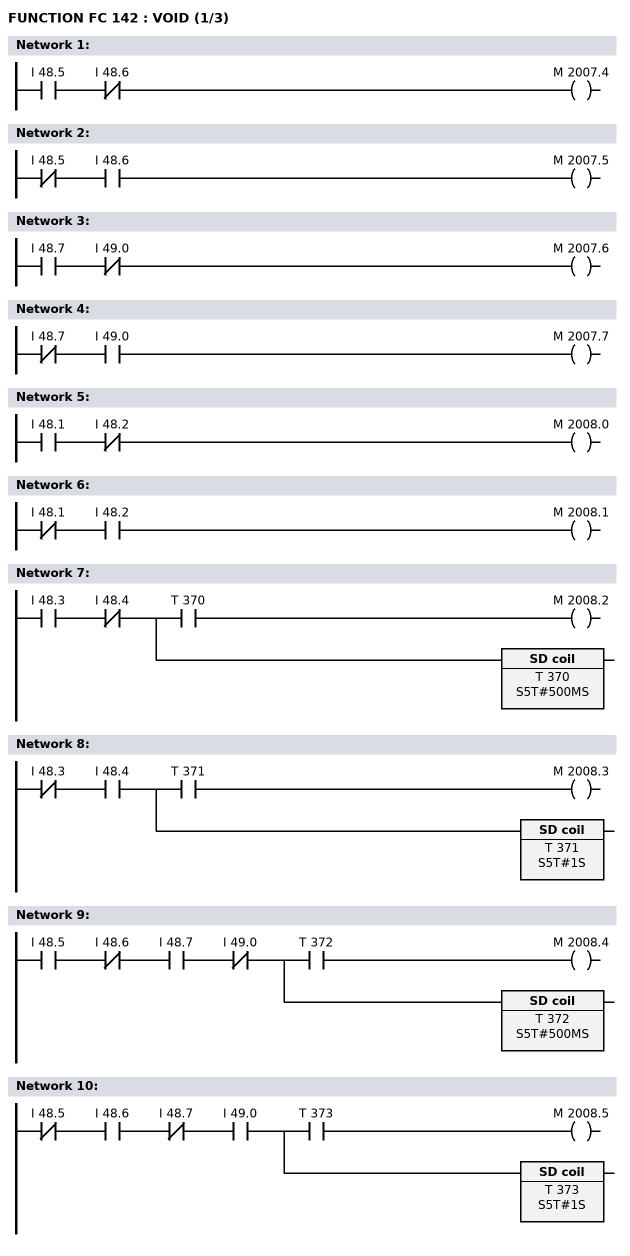

      A     I     48.5;
      AN    I     48.6;
      =     M   2007.4;
NETWORK
TITLE =

      AN    I     48.5;
      A     I     48.6;
      =     M   2007.5;
NETWORK
TITLE =

      A     I     48.7;
      AN    I     49.0;
      =     M   2007.6;
NETWORK
TITLE =

      AN    I     48.7;
      A     I     49.0;
      =     M   2007.7;
NETWORK
TITLE =

      A     I     48.1;
      AN    I     48.2;
      =     M   2008.0;
NETWORK
TITLE =

      AN    I     48.1;
      A     I     48.2;
      =     M   2008.1;
NETWORK
TITLE =

      A     I     48.3;
      AN    I     48.4;
      =     L      0.0;
      A     L      0.0;
      A     T    370;
      =     M   2008.2;
      A     L      0.0;
      BLD   102;
      L     S5T#500MS;
      SD    T    370;
NETWORK
TITLE =

      AN    I     48.3;
      A     I     48.4;
      =     L      0.0;
      A     L      0.0;
      A     T    371;
      =     M   2008.3;
      A     L      0.0;
      BLD   102;
      L     S5T#1S;
      SD    T    371;
NETWORK
TITLE =

      A     I     48.5;
      AN    I     48.6;
      A     I     48.7;
      AN    I     49.0;
      =     L      0.0;
      A     L      0.0;
      A     T    372;
      =     M   2008.4;
      A     L      0.0;
      BLD   102;
      L     S5T#500MS;
      SD    T    372;
NETWORK
TITLE =

      AN    I     48.5;
      A     I     48.6;
      AN    I     48.7;
      A     I     49.0;
      =     L      0.0;
      A     L      0.0;
      A     T    373;
      =     M   2008.5;
      A     L      0.0;
      BLD   102;
      L     S5T#1S;
      SD    T    373;
NETWORK
TITLE =
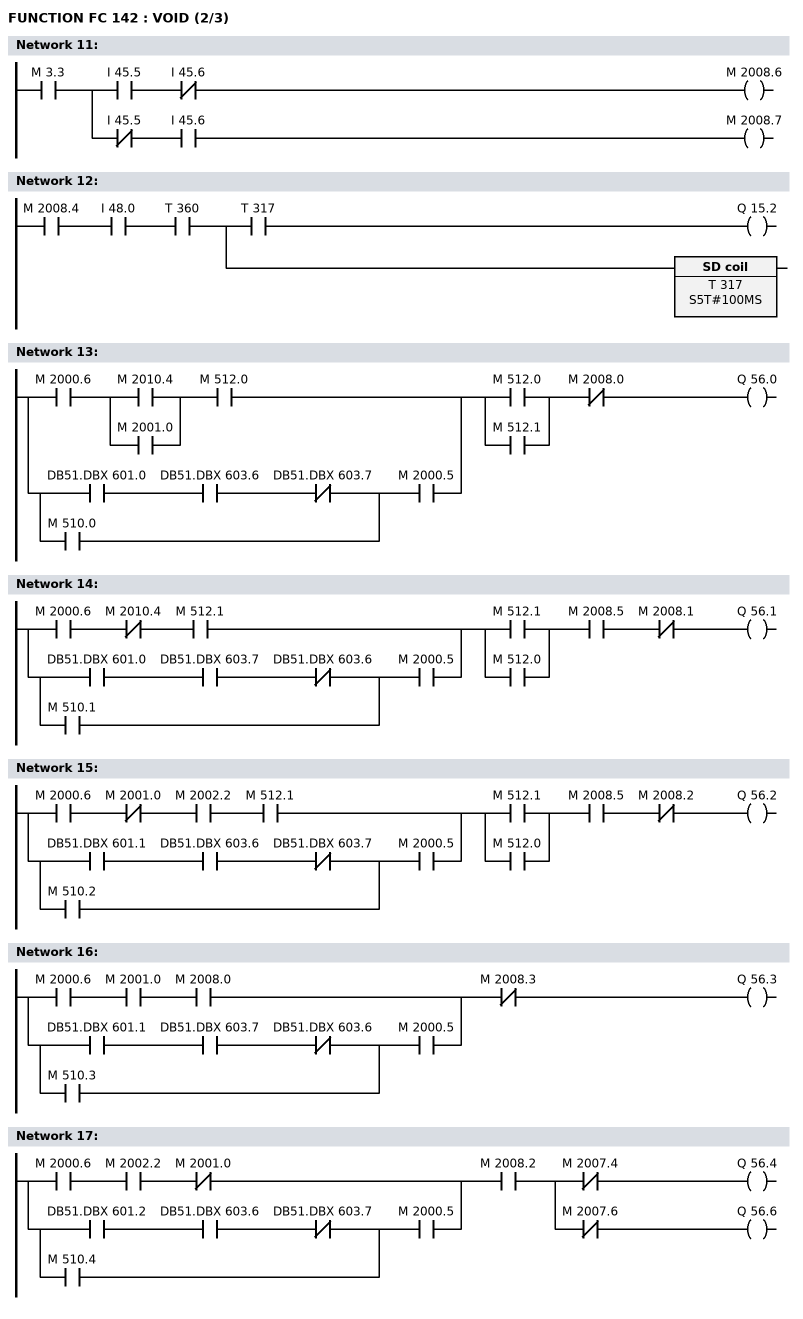

      A     M      3.3;
      =     L      0.0;
      A     L      0.0;
      A     I     45.5;
      AN    I     45.6;
      =     M   2008.6;
      A     L      0.0;
      AN    I     45.5;
      A     I     45.6;
      =     M   2008.7;
NETWORK
TITLE =

      A     M   2008.4;
      A     I     48.0;
      A     T    360;
      =     L      0.0;
      A     L      0.0;
      A     T    317;
      =     Q     15.2;
      A     L      0.0;
      BLD   102;
      L     S5T#100MS;
      SD    T    317;
NETWORK
TITLE =

      A(    ;
      A     M   2000.6;
      A(    ;
      O     M   2010.4;
      O     M   2001.0;
      )     ;
      A     M    512.0;
      O     ;
      A(    ;
      A     DB51.DBX  601.0;
      A     DB51.DBX  603.6;
      AN    DB51.DBX  603.7;
      O     M    510.0;
      )     ;
      A     M   2000.5;
      )     ;
      A(    ;
      O     M    512.0;
      O     M    512.1;
      )     ;
      AN    M   2008.0;
      =     Q     56.0;
NETWORK
TITLE =

      A(    ;
      A     M   2000.6;
      AN    M   2010.4;
      A     M    512.1;
      O     ;
      A(    ;
      A     DB51.DBX  601.0;
      A     DB51.DBX  603.7;
      AN    DB51.DBX  603.6;
      O     M    510.1;
      )     ;
      A     M   2000.5;
      )     ;
      A(    ;
      O     M    512.1;
      O     M    512.0;
      )     ;
      A     M   2008.5;
      AN    M   2008.1;
      =     Q     56.1;
NETWORK
TITLE =

      A(    ;
      A     M   2000.6;
      AN    M   2001.0;
      A     M   2002.2;
      A     M    512.1;
      O     ;
      A(    ;
      A     DB51.DBX  601.1;
      A     DB51.DBX  603.6;
      AN    DB51.DBX  603.7;
      O     M    510.2;
      )     ;
      A     M   2000.5;
      )     ;
      A(    ;
      O     M    512.1;
      O     M    512.0;
      )     ;
      A     M   2008.5;
      AN    M   2008.2;
      =     Q     56.2;
NETWORK
TITLE =

      A(    ;
      A     M   2000.6;
      A     M   2001.0;
      A     M   2008.0;
      O     ;
      A(    ;
      A     DB51.DBX  601.1;
      A     DB51.DBX  603.7;
      AN    DB51.DBX  603.6;
      O     M    510.3;
      )     ;
      A     M   2000.5;
      )     ;
      AN    M   2008.3;
      =     Q     56.3;
NETWORK
TITLE =

      A(    ;
      A     M   2000.6;
      A     M   2002.2;
      AN    M   2001.0;
      O     ;
      A(    ;
      A     DB51.DBX  601.2;
      A     DB51.DBX  603.6;
      AN    DB51.DBX  603.7;
      O     M    510.4;
      )     ;
      A     M   2000.5;
      )     ;
      A     M   2008.2;
      =     L      0.0;
      A     L      0.0;
      AN    M   2007.4;
      =     Q     56.4;
      A     L      0.0;
      AN    M   2007.6;
      =     Q     56.6;
NETWORK
TITLE =
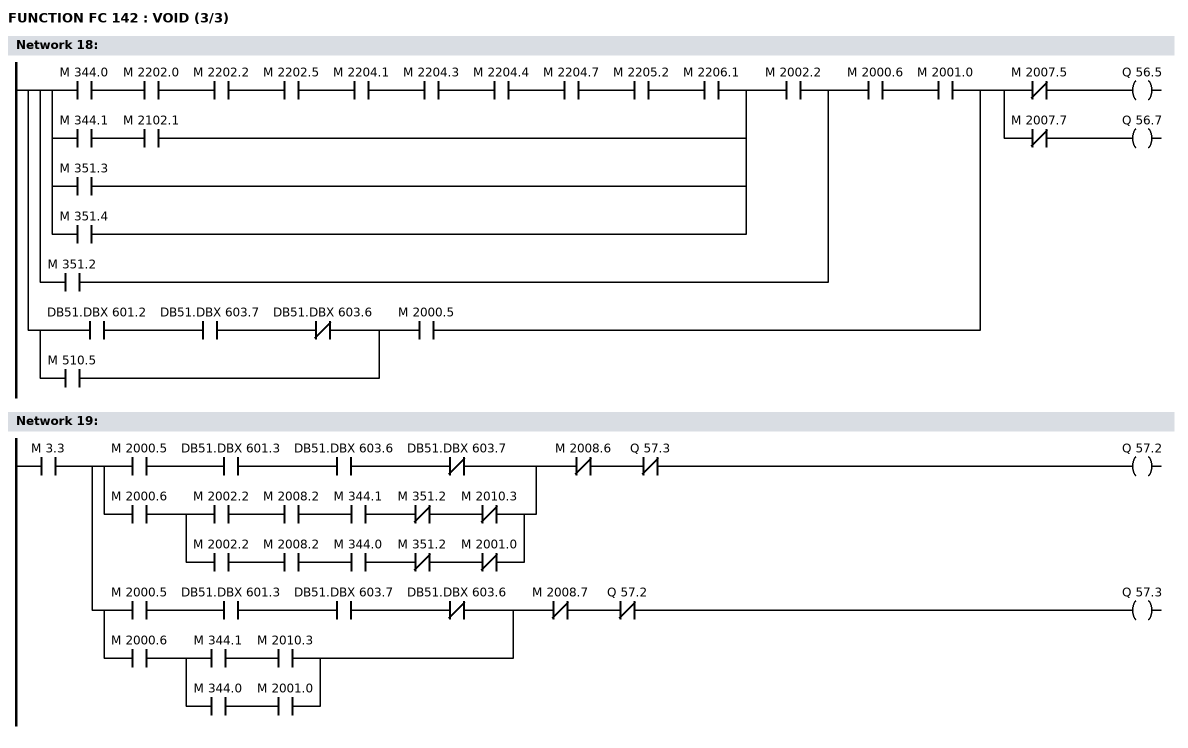

      A(    ;
      A(    ;
      A     M    344.0;
      A     M   2202.0;
      A     M   2202.2;
      A     M   2202.5;
      A     M   2204.1;
      A     M   2204.3;
      A     M   2204.4;
      A     M   2204.7;
      A     M   2205.2;
      A     M   2206.1;
      O     ;
      A     M    344.1;
      A     M   2102.1;
      O     M    351.3;
      O     M    351.4;
      )     ;
      A     M   2002.2;
      O     M    351.2;
      )     ;
      A     M   2000.6;
      A     M   2001.0;
      O     ;
      A(    ;
      A     DB51.DBX  601.2;
      A     DB51.DBX  603.7;
      AN    DB51.DBX  603.6;
      O     M    510.5;
      )     ;
      A     M   2000.5;
      =     L      0.0;
      A     L      0.0;
      AN    M   2007.5;
      =     Q     56.5;
      A     L      0.0;
      AN    M   2007.7;
      =     Q     56.7;
NETWORK
TITLE =

      A     M      3.3;
      =     L      0.0;
      A     L      0.0;
      A(    ;
      A     M   2000.5;
      A     DB51.DBX  601.3;
      A     DB51.DBX  603.6;
      AN    DB51.DBX  603.7;
      O     ;
      A     M   2000.6;
      A(    ;
      A     M   2002.2;
      A     M   2008.2;
      A     M    344.1;
      AN    M    351.2;
      AN    M   2010.3;
      O     ;
      A     M   2002.2;
      A     M   2008.2;
      A     M    344.0;
      AN    M    351.2;
      AN    M   2001.0;
      )     ;
      )     ;
      AN    M   2008.6;
      AN    Q     57.3;
      =     Q     57.2;
      A     L      0.0;
      A(    ;
      A     M   2000.5;
      A     DB51.DBX  601.3;
      A     DB51.DBX  603.7;
      AN    DB51.DBX  603.6;
      O     ;
      A     M   2000.6;
      A(    ;
      A     M    344.1;
      A     M   2010.3;
      O     ;
      A     M    344.0;
      A     M   2001.0;
      )     ;
      )     ;
      AN    M   2008.7;
      AN    Q     57.2;
      =     Q     57.3;
END_FUNCTION

FUNCTION_BLOCK FB 143
TITLE =
VERSION : 0.1


VAR
  S704_LM_DC_PIN : FB 424;
  S704_LM_DC_1ST_CLAMP1 : FB 424;
  S704_LM_DC_1ST_CLAMP2 : FB 424;
  S704_LM_DC_1ST_CLAMP3 : FB 424;
  S704_LM_DC_1ST_CLAMP4 : FB 424;
  S704_LM_DC_2ND_CLAMP1 : FB 424;
  S704_LM_DC_2ND_CLAMP2 : FB 424;
  S704_LM_DC_2ND_CLAMP3 : FB 424;
  S704_LM_DC_2ND_CLAMP4 : FB 424;
  S704_LM_DC_2ND_CLAMP5 : FB 424;
  S704_LM_DC_STK_PIN : FB 424;
  S704_LM_DC_OTR_CLAMP : FB 424;
  S704_LM_DC_ASSY_CLAMP : FB 424;
  S704_LM_DC_FF_PIN : FB 424;
  S704_LM_DC_FF_CLAMP : FB 424;
  S704_LM_DC_2ND_CLAMP6 : FB 424;
  S704_LM_DC_2ND_CLAMP7 : FB 424;
  S704_LM_DC_1ST_CLAMP5 : FB 424;
END_VAR
BEGIN
NETWORK
TITLE =
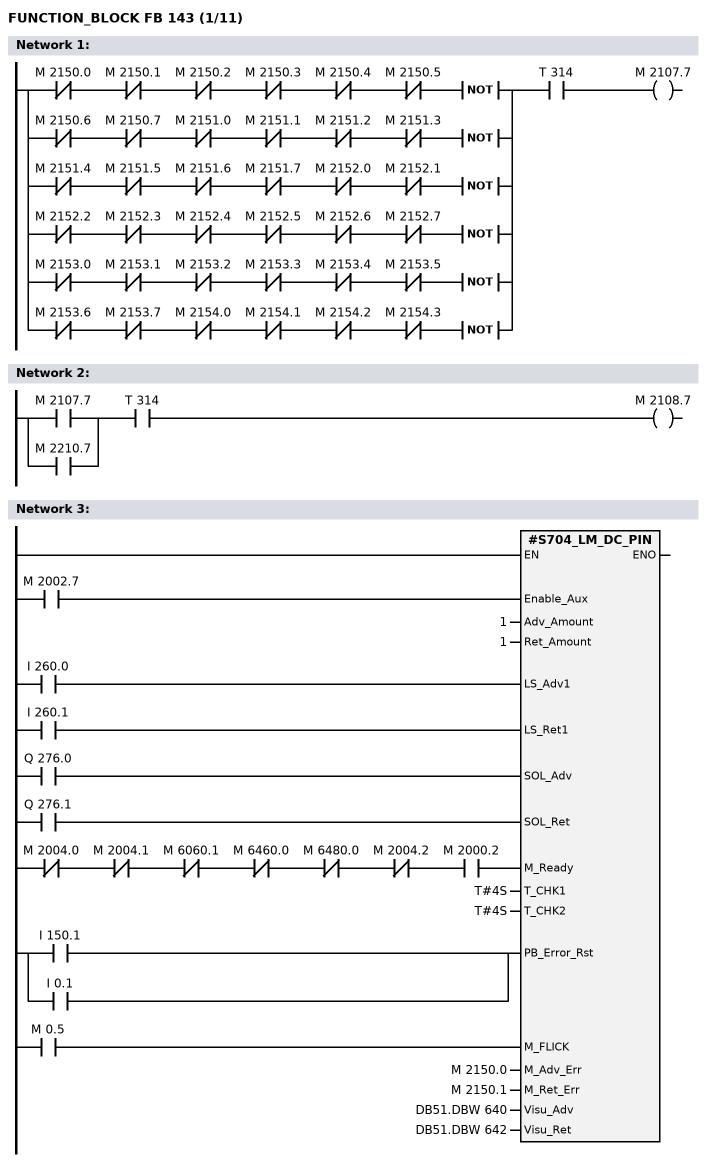

      A(    ;
      AN    M   2150.0;
      AN    M   2150.1;
      AN    M   2150.2;
      AN    M   2150.3;
      AN    M   2150.4;
      AN    M   2150.5;
      NOT   ;
      O(    ;
      AN    M   2150.6;
      AN    M   2150.7;
      AN    M   2151.0;
      AN    M   2151.1;
      AN    M   2151.2;
      AN    M   2151.3;
      NOT   ;
      )     ;
      O(    ;
      AN    M   2151.4;
      AN    M   2151.5;
      AN    M   2151.6;
      AN    M   2151.7;
      AN    M   2152.0;
      AN    M   2152.1;
      NOT   ;
      )     ;
      O(    ;
      AN    M   2152.2;
      AN    M   2152.3;
      AN    M   2152.4;
      AN    M   2152.5;
      AN    M   2152.6;
      AN    M   2152.7;
      NOT   ;
      )     ;
      O(    ;
      AN    M   2153.0;
      AN    M   2153.1;
      AN    M   2153.2;
      AN    M   2153.3;
      AN    M   2153.4;
      AN    M   2153.5;
      NOT   ;
      )     ;
      O(    ;
      AN    M   2153.6;
      AN    M   2153.7;
      AN    M   2154.0;
      AN    M   2154.1;
      AN    M   2154.2;
      AN    M   2154.3;
      NOT   ;
      )     ;
      )     ;
      A     T    314;
      =     M   2107.7;
NETWORK
TITLE =

      A(    ;
      O     M   2107.7;
      O     M   2210.7;
      )     ;
      A     T    314;
      =     M   2108.7;
NETWORK
TITLE =

      A     M   2002.7;
      =     L      0.0;
      BLD   103;
      A     I    260.0;
      =     L      0.1;
      BLD   103;
      A     I    260.1;
      =     L      0.2;
      BLD   103;
      A     Q    276.0;
      =     L      1.1;
      BLD   103;
      A     Q    276.1;
      =     L      1.2;
      BLD   103;
      AN    M   2004.0;
      AN    M   2004.1;
      AN    M   6060.1;
      AN    M   6460.0;
      AN    M   6480.0;
      AN    M   2004.2;
      A     M   2000.2;
      =     L      1.3;
      BLD   103;
      A(    ;
      O     I    150.1;
      O     I      0.1;
      )     ;
      =     L      1.5;
      BLD   103;
      A     M      0.5;
      =     L      1.6;
      BLD   103;
      CALL #S704_LM_DC_PIN (
           Enable_Aux               := L      0.0,
           Adv_Amount               := 1,
           Ret_Amount               := 1,
           LS_Adv1                  := L      0.1,
           LS_Ret1                  := L      0.2,
           SOL_Adv                  := L      1.1,
           SOL_Ret                  := L      1.2,
           M_Ready                  := L      1.3,
           T_CHK1                   := T#4S,
           T_CHK2                   := T#4S,
           PB_Error_Rst             := L      1.5,
           M_FLICK                  := L      1.6,
           M_Adv_Err                := M   2150.0,
           M_Ret_Err                := M   2150.1,
           Visu_Adv                 := DB51.DBW  640,
           Visu_Ret                 := DB51.DBW  642);
      NOP   0;
NETWORK
TITLE =
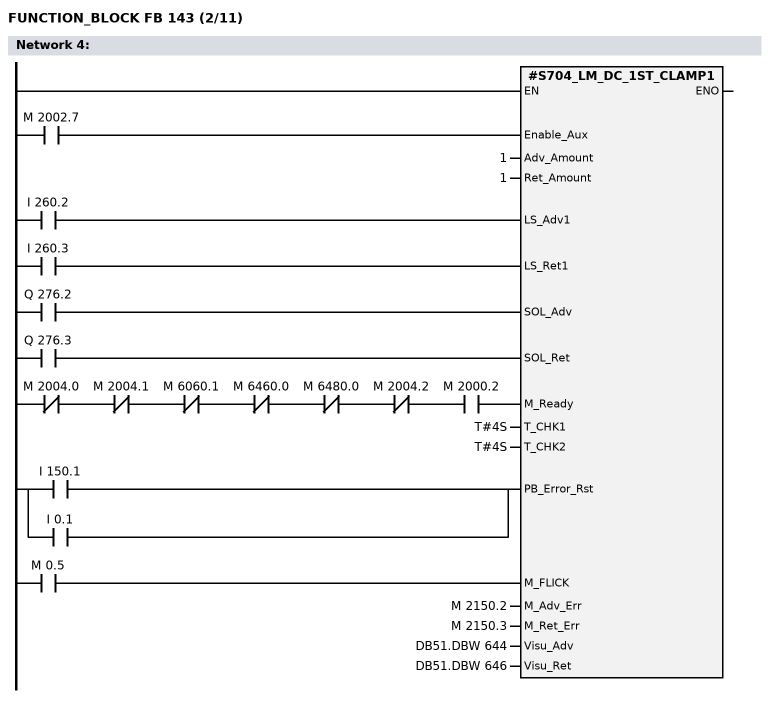

      A     M   2002.7;
      =     L      0.0;
      BLD   103;
      A     I    260.2;
      =     L      0.1;
      BLD   103;
      A     I    260.3;
      =     L      0.2;
      BLD   103;
      A     Q    276.2;
      =     L      1.1;
      BLD   103;
      A     Q    276.3;
      =     L      1.2;
      BLD   103;
      AN    M   2004.0;
      AN    M   2004.1;
      AN    M   6060.1;
      AN    M   6460.0;
      AN    M   6480.0;
      AN    M   2004.2;
      A     M   2000.2;
      =     L      1.3;
      BLD   103;
      A(    ;
      O     I    150.1;
      O     I      0.1;
      )     ;
      =     L      1.5;
      BLD   103;
      A     M      0.5;
      =     L      1.6;
      BLD   103;
      CALL #S704_LM_DC_1ST_CLAMP1 (
           Enable_Aux               := L      0.0,
           Adv_Amount               := 1,
           Ret_Amount               := 1,
           LS_Adv1                  := L      0.1,
           LS_Ret1                  := L      0.2,
           SOL_Adv                  := L      1.1,
           SOL_Ret                  := L      1.2,
           M_Ready                  := L      1.3,
           T_CHK1                   := T#4S,
           T_CHK2                   := T#4S,
           PB_Error_Rst             := L      1.5,
           M_FLICK                  := L      1.6,
           M_Adv_Err                := M   2150.2,
           M_Ret_Err                := M   2150.3,
           Visu_Adv                 := DB51.DBW  644,
           Visu_Ret                 := DB51.DBW  646);
      NOP   0;
NETWORK
TITLE =
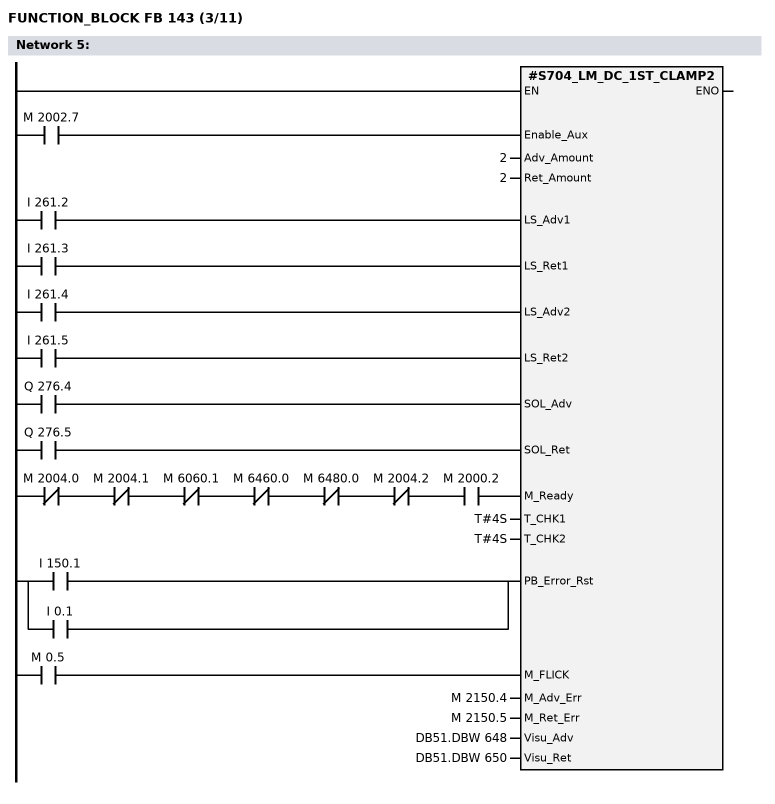

      A     M   2002.7;
      =     L      0.0;
      BLD   103;
      A     I    261.2;
      =     L      0.1;
      BLD   103;
      A     I    261.3;
      =     L      0.2;
      BLD   103;
      A     I    261.4;
      =     L      0.3;
      BLD   103;
      A     I    261.5;
      =     L      0.4;
      BLD   103;
      A     Q    276.4;
      =     L      1.1;
      BLD   103;
      A     Q    276.5;
      =     L      1.2;
      BLD   103;
      AN    M   2004.0;
      AN    M   2004.1;
      AN    M   6060.1;
      AN    M   6460.0;
      AN    M   6480.0;
      AN    M   2004.2;
      A     M   2000.2;
      =     L      1.3;
      BLD   103;
      A(    ;
      O     I    150.1;
      O     I      0.1;
      )     ;
      =     L      1.5;
      BLD   103;
      A     M      0.5;
      =     L      1.6;
      BLD   103;
      CALL #S704_LM_DC_1ST_CLAMP2 (
           Enable_Aux               := L      0.0,
           Adv_Amount               := 2,
           Ret_Amount               := 2,
           LS_Adv1                  := L      0.1,
           LS_Ret1                  := L      0.2,
           LS_Adv2                  := L      0.3,
           LS_Ret2                  := L      0.4,
           SOL_Adv                  := L      1.1,
           SOL_Ret                  := L      1.2,
           M_Ready                  := L      1.3,
           T_CHK1                   := T#4S,
           T_CHK2                   := T#4S,
           PB_Error_Rst             := L      1.5,
           M_FLICK                  := L      1.6,
           M_Adv_Err                := M   2150.4,
           M_Ret_Err                := M   2150.5,
           Visu_Adv                 := DB51.DBW  648,
           Visu_Ret                 := DB51.DBW  650);
      NOP   0;
NETWORK
TITLE =
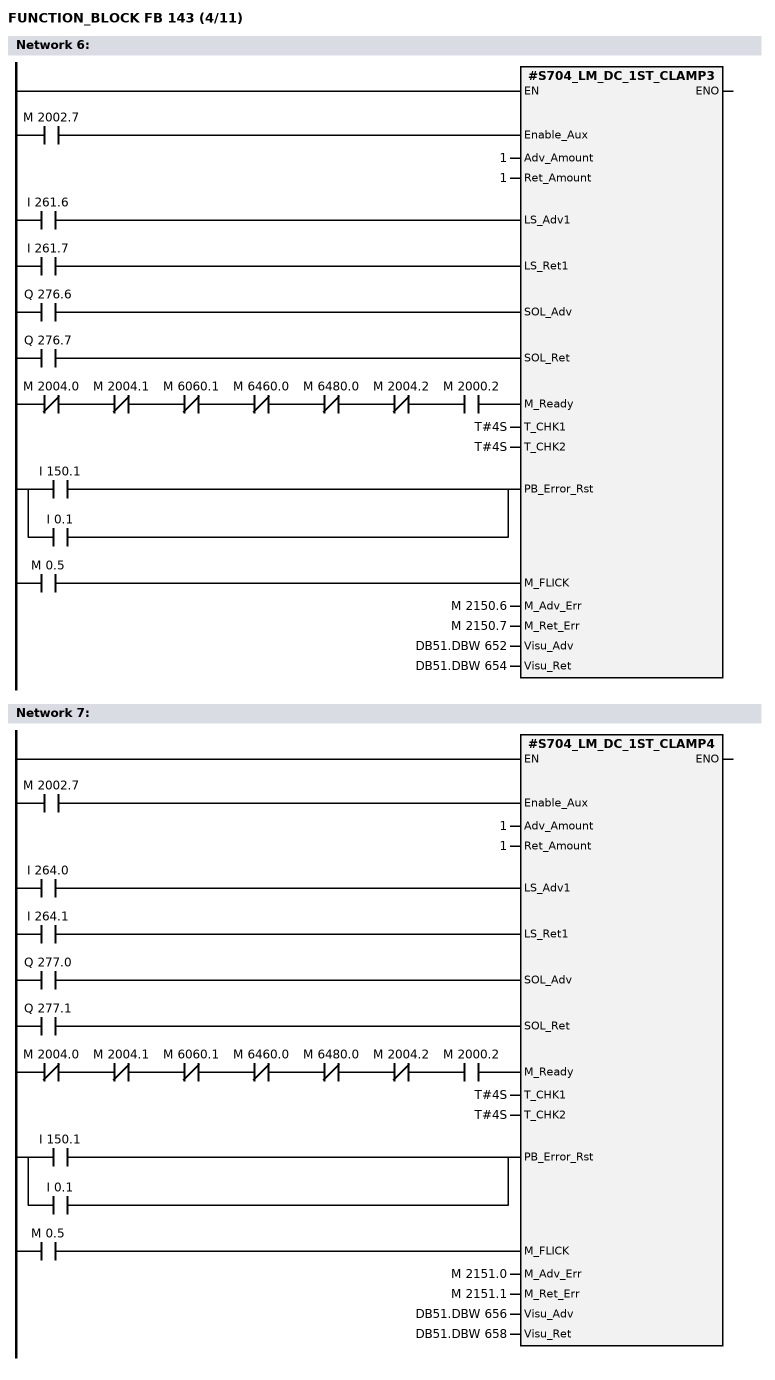

      A     M   2002.7;
      =     L      0.0;
      BLD   103;
      A     I    261.6;
      =     L      0.1;
      BLD   103;
      A     I    261.7;
      =     L      0.2;
      BLD   103;
      A     Q    276.6;
      =     L      1.1;
      BLD   103;
      A     Q    276.7;
      =     L      1.2;
      BLD   103;
      AN    M   2004.0;
      AN    M   2004.1;
      AN    M   6060.1;
      AN    M   6460.0;
      AN    M   6480.0;
      AN    M   2004.2;
      A     M   2000.2;
      =     L      1.3;
      BLD   103;
      A(    ;
      O     I    150.1;
      O     I      0.1;
      )     ;
      =     L      1.5;
      BLD   103;
      A     M      0.5;
      =     L      1.6;
      BLD   103;
      CALL #S704_LM_DC_1ST_CLAMP3 (
           Enable_Aux               := L      0.0,
           Adv_Amount               := 1,
           Ret_Amount               := 1,
           LS_Adv1                  := L      0.1,
           LS_Ret1                  := L      0.2,
           SOL_Adv                  := L      1.1,
           SOL_Ret                  := L      1.2,
           M_Ready                  := L      1.3,
           T_CHK1                   := T#4S,
           T_CHK2                   := T#4S,
           PB_Error_Rst             := L      1.5,
           M_FLICK                  := L      1.6,
           M_Adv_Err                := M   2150.6,
           M_Ret_Err                := M   2150.7,
           Visu_Adv                 := DB51.DBW  652,
           Visu_Ret                 := DB51.DBW  654);
      NOP   0;
NETWORK
TITLE =

      A     M   2002.7;
      =     L      0.0;
      BLD   103;
      A     I    264.0;
      =     L      0.1;
      BLD   103;
      A     I    264.1;
      =     L      0.2;
      BLD   103;
      A     Q    277.0;
      =     L      1.1;
      BLD   103;
      A     Q    277.1;
      =     L      1.2;
      BLD   103;
      AN    M   2004.0;
      AN    M   2004.1;
      AN    M   6060.1;
      AN    M   6460.0;
      AN    M   6480.0;
      AN    M   2004.2;
      A     M   2000.2;
      =     L      1.3;
      BLD   103;
      A(    ;
      O     I    150.1;
      O     I      0.1;
      )     ;
      =     L      1.5;
      BLD   103;
      A     M      0.5;
      =     L      1.6;
      BLD   103;
      CALL #S704_LM_DC_1ST_CLAMP4 (
           Enable_Aux               := L      0.0,
           Adv_Amount               := 1,
           Ret_Amount               := 1,
           LS_Adv1                  := L      0.1,
           LS_Ret1                  := L      0.2,
           SOL_Adv                  := L      1.1,
           SOL_Ret                  := L      1.2,
           M_Ready                  := L      1.3,
           T_CHK1                   := T#4S,
           T_CHK2                   := T#4S,
           PB_Error_Rst             := L      1.5,
           M_FLICK                  := L      1.6,
           M_Adv_Err                := M   2151.0,
           M_Ret_Err                := M   2151.1,
           Visu_Adv                 := DB51.DBW  656,
           Visu_Ret                 := DB51.DBW  658);
      NOP   0;
NETWORK
TITLE =
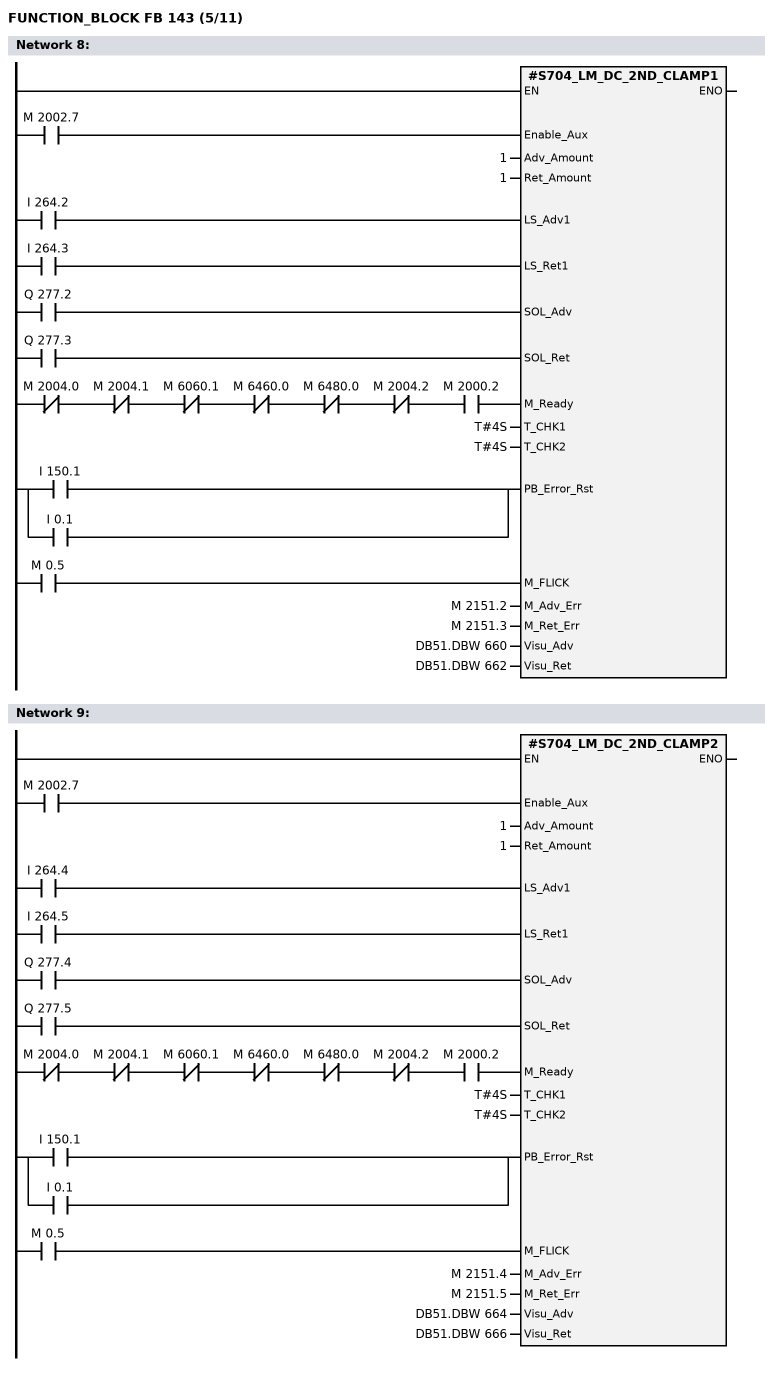

      A     M   2002.7;
      =     L      0.0;
      BLD   103;
      A     I    264.2;
      =     L      0.1;
      BLD   103;
      A     I    264.3;
      =     L      0.2;
      BLD   103;
      A     Q    277.2;
      =     L      1.1;
      BLD   103;
      A     Q    277.3;
      =     L      1.2;
      BLD   103;
      AN    M   2004.0;
      AN    M   2004.1;
      AN    M   6060.1;
      AN    M   6460.0;
      AN    M   6480.0;
      AN    M   2004.2;
      A     M   2000.2;
      =     L      1.3;
      BLD   103;
      A(    ;
      O     I    150.1;
      O     I      0.1;
      )     ;
      =     L      1.5;
      BLD   103;
      A     M      0.5;
      =     L      1.6;
      BLD   103;
      CALL #S704_LM_DC_2ND_CLAMP1 (
           Enable_Aux               := L      0.0,
           Adv_Amount               := 1,
           Ret_Amount               := 1,
           LS_Adv1                  := L      0.1,
           LS_Ret1                  := L      0.2,
           SOL_Adv                  := L      1.1,
           SOL_Ret                  := L      1.2,
           M_Ready                  := L      1.3,
           T_CHK1                   := T#4S,
           T_CHK2                   := T#4S,
           PB_Error_Rst             := L      1.5,
           M_FLICK                  := L      1.6,
           M_Adv_Err                := M   2151.2,
           M_Ret_Err                := M   2151.3,
           Visu_Adv                 := DB51.DBW  660,
           Visu_Ret                 := DB51.DBW  662);
      NOP   0;
NETWORK
TITLE =

      A     M   2002.7;
      =     L      0.0;
      BLD   103;
      A     I    264.4;
      =     L      0.1;
      BLD   103;
      A     I    264.5;
      =     L      0.2;
      BLD   103;
      A     Q    277.4;
      =     L      1.1;
      BLD   103;
      A     Q    277.5;
      =     L      1.2;
      BLD   103;
      AN    M   2004.0;
      AN    M   2004.1;
      AN    M   6060.1;
      AN    M   6460.0;
      AN    M   6480.0;
      AN    M   2004.2;
      A     M   2000.2;
      =     L      1.3;
      BLD   103;
      A(    ;
      O     I    150.1;
      O     I      0.1;
      )     ;
      =     L      1.5;
      BLD   103;
      A     M      0.5;
      =     L      1.6;
      BLD   103;
      CALL #S704_LM_DC_2ND_CLAMP2 (
           Enable_Aux               := L      0.0,
           Adv_Amount               := 1,
           Ret_Amount               := 1,
           LS_Adv1                  := L      0.1,
           LS_Ret1                  := L      0.2,
           SOL_Adv                  := L      1.1,
           SOL_Ret                  := L      1.2,
           M_Ready                  := L      1.3,
           T_CHK1                   := T#4S,
           T_CHK2                   := T#4S,
           PB_Error_Rst             := L      1.5,
           M_FLICK                  := L      1.6,
           M_Adv_Err                := M   2151.4,
           M_Ret_Err                := M   2151.5,
           Visu_Adv                 := DB51.DBW  664,
           Visu_Ret                 := DB51.DBW  666);
      NOP   0;
NETWORK
TITLE =
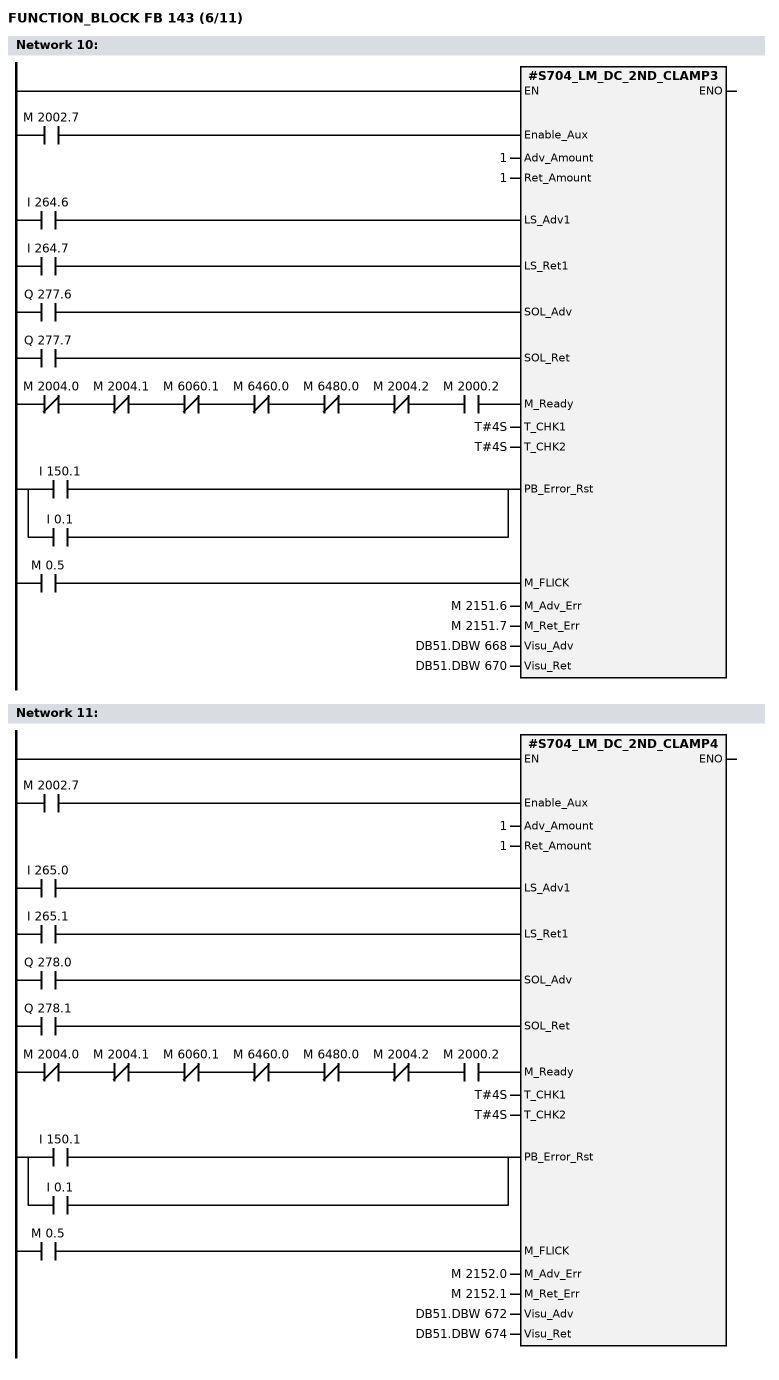

      A     M   2002.7;
      =     L      0.0;
      BLD   103;
      A     I    264.6;
      =     L      0.1;
      BLD   103;
      A     I    264.7;
      =     L      0.2;
      BLD   103;
      A     Q    277.6;
      =     L      1.1;
      BLD   103;
      A     Q    277.7;
      =     L      1.2;
      BLD   103;
      AN    M   2004.0;
      AN    M   2004.1;
      AN    M   6060.1;
      AN    M   6460.0;
      AN    M   6480.0;
      AN    M   2004.2;
      A     M   2000.2;
      =     L      1.3;
      BLD   103;
      A(    ;
      O     I    150.1;
      O     I      0.1;
      )     ;
      =     L      1.5;
      BLD   103;
      A     M      0.5;
      =     L      1.6;
      BLD   103;
      CALL #S704_LM_DC_2ND_CLAMP3 (
           Enable_Aux               := L      0.0,
           Adv_Amount               := 1,
           Ret_Amount               := 1,
           LS_Adv1                  := L      0.1,
           LS_Ret1                  := L      0.2,
           SOL_Adv                  := L      1.1,
           SOL_Ret                  := L      1.2,
           M_Ready                  := L      1.3,
           T_CHK1                   := T#4S,
           T_CHK2                   := T#4S,
           PB_Error_Rst             := L      1.5,
           M_FLICK                  := L      1.6,
           M_Adv_Err                := M   2151.6,
           M_Ret_Err                := M   2151.7,
           Visu_Adv                 := DB51.DBW  668,
           Visu_Ret                 := DB51.DBW  670);
      NOP   0;
NETWORK
TITLE =

      A     M   2002.7;
      =     L      0.0;
      BLD   103;
      A     I    265.0;
      =     L      0.1;
      BLD   103;
      A     I    265.1;
      =     L      0.2;
      BLD   103;
      A     Q    278.0;
      =     L      1.1;
      BLD   103;
      A     Q    278.1;
      =     L      1.2;
      BLD   103;
      AN    M   2004.0;
      AN    M   2004.1;
      AN    M   6060.1;
      AN    M   6460.0;
      AN    M   6480.0;
      AN    M   2004.2;
      A     M   2000.2;
      =     L      1.3;
      BLD   103;
      A(    ;
      O     I    150.1;
      O     I      0.1;
      )     ;
      =     L      1.5;
      BLD   103;
      A     M      0.5;
      =     L      1.6;
      BLD   103;
      CALL #S704_LM_DC_2ND_CLAMP4 (
           Enable_Aux               := L      0.0,
           Adv_Amount               := 1,
           Ret_Amount               := 1,
           LS_Adv1                  := L      0.1,
           LS_Ret1                  := L      0.2,
           SOL_Adv                  := L      1.1,
           SOL_Ret                  := L      1.2,
           M_Ready                  := L      1.3,
           T_CHK1                   := T#4S,
           T_CHK2                   := T#4S,
           PB_Error_Rst             := L      1.5,
           M_FLICK                  := L      1.6,
           M_Adv_Err                := M   2152.0,
           M_Ret_Err                := M   2152.1,
           Visu_Adv                 := DB51.DBW  672,
           Visu_Ret                 := DB51.DBW  674);
      NOP   0;
NETWORK
TITLE =
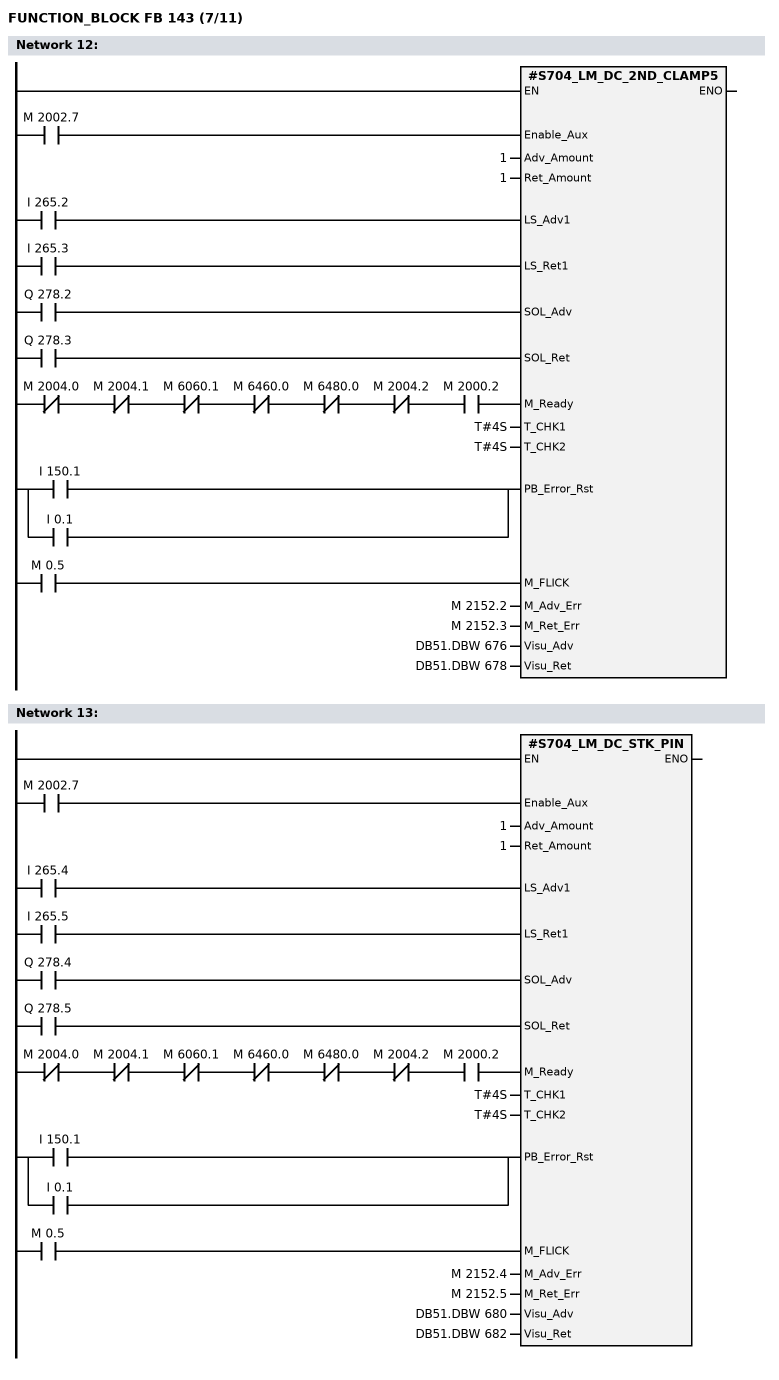

      A     M   2002.7;
      =     L      0.0;
      BLD   103;
      A     I    265.2;
      =     L      0.1;
      BLD   103;
      A     I    265.3;
      =     L      0.2;
      BLD   103;
      A     Q    278.2;
      =     L      1.1;
      BLD   103;
      A     Q    278.3;
      =     L      1.2;
      BLD   103;
      AN    M   2004.0;
      AN    M   2004.1;
      AN    M   6060.1;
      AN    M   6460.0;
      AN    M   6480.0;
      AN    M   2004.2;
      A     M   2000.2;
      =     L      1.3;
      BLD   103;
      A(    ;
      O     I    150.1;
      O     I      0.1;
      )     ;
      =     L      1.5;
      BLD   103;
      A     M      0.5;
      =     L      1.6;
      BLD   103;
      CALL #S704_LM_DC_2ND_CLAMP5 (
           Enable_Aux               := L      0.0,
           Adv_Amount               := 1,
           Ret_Amount               := 1,
           LS_Adv1                  := L      0.1,
           LS_Ret1                  := L      0.2,
           SOL_Adv                  := L      1.1,
           SOL_Ret                  := L      1.2,
           M_Ready                  := L      1.3,
           T_CHK1                   := T#4S,
           T_CHK2                   := T#4S,
           PB_Error_Rst             := L      1.5,
           M_FLICK                  := L      1.6,
           M_Adv_Err                := M   2152.2,
           M_Ret_Err                := M   2152.3,
           Visu_Adv                 := DB51.DBW  676,
           Visu_Ret                 := DB51.DBW  678);
      NOP   0;
NETWORK
TITLE =

      A     M   2002.7;
      =     L      0.0;
      BLD   103;
      A     I    265.4;
      =     L      0.1;
      BLD   103;
      A     I    265.5;
      =     L      0.2;
      BLD   103;
      A     Q    278.4;
      =     L      1.1;
      BLD   103;
      A     Q    278.5;
      =     L      1.2;
      BLD   103;
      AN    M   2004.0;
      AN    M   2004.1;
      AN    M   6060.1;
      AN    M   6460.0;
      AN    M   6480.0;
      AN    M   2004.2;
      A     M   2000.2;
      =     L      1.3;
      BLD   103;
      A(    ;
      O     I    150.1;
      O     I      0.1;
      )     ;
      =     L      1.5;
      BLD   103;
      A     M      0.5;
      =     L      1.6;
      BLD   103;
      CALL #S704_LM_DC_STK_PIN (
           Enable_Aux               := L      0.0,
           Adv_Amount               := 1,
           Ret_Amount               := 1,
           LS_Adv1                  := L      0.1,
           LS_Ret1                  := L      0.2,
           SOL_Adv                  := L      1.1,
           SOL_Ret                  := L      1.2,
           M_Ready                  := L      1.3,
           T_CHK1                   := T#4S,
           T_CHK2                   := T#4S,
           PB_Error_Rst             := L      1.5,
           M_FLICK                  := L      1.6,
           M_Adv_Err                := M   2152.4,
           M_Ret_Err                := M   2152.5,
           Visu_Adv                 := DB51.DBW  680,
           Visu_Ret                 := DB51.DBW  682);
      NOP   0;
NETWORK
TITLE =
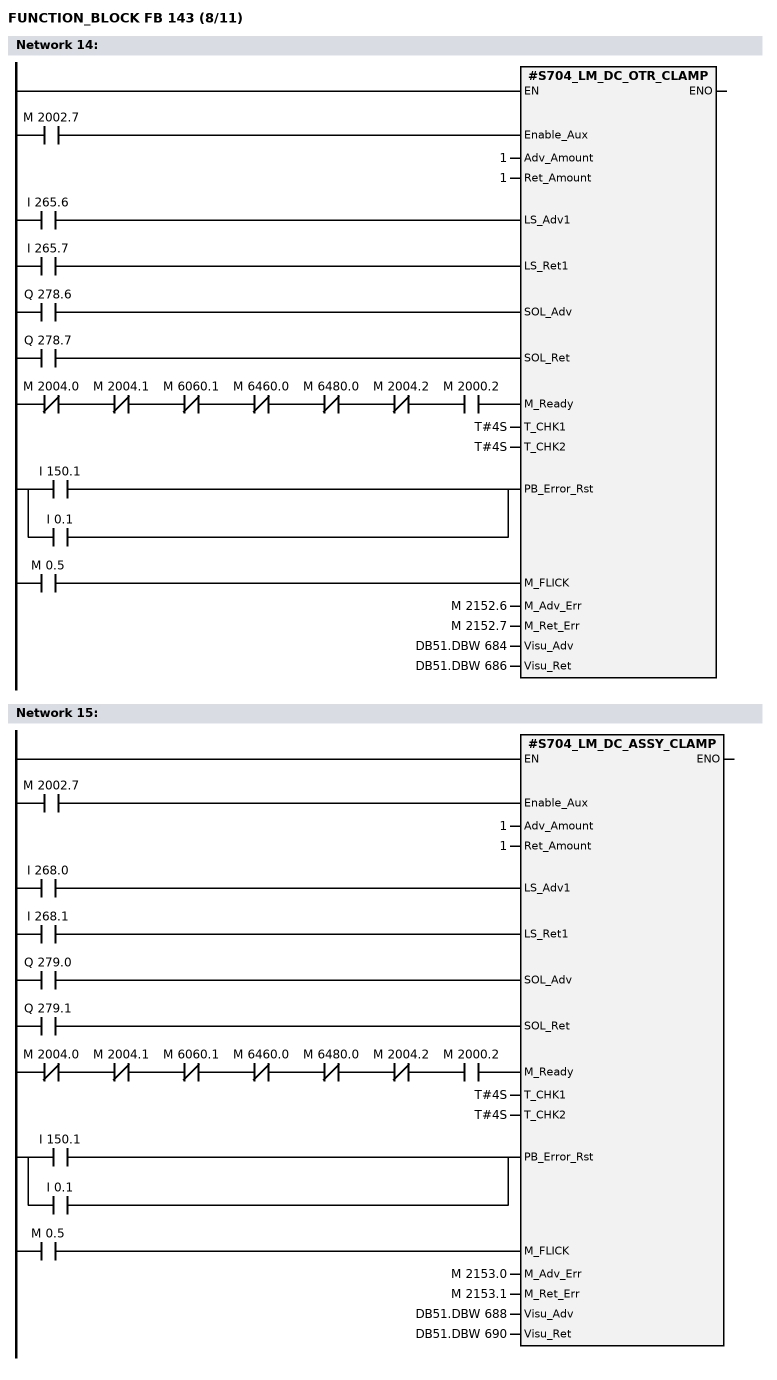

      A     M   2002.7;
      =     L      0.0;
      BLD   103;
      A     I    265.6;
      =     L      0.1;
      BLD   103;
      A     I    265.7;
      =     L      0.2;
      BLD   103;
      A     Q    278.6;
      =     L      1.1;
      BLD   103;
      A     Q    278.7;
      =     L      1.2;
      BLD   103;
      AN    M   2004.0;
      AN    M   2004.1;
      AN    M   6060.1;
      AN    M   6460.0;
      AN    M   6480.0;
      AN    M   2004.2;
      A     M   2000.2;
      =     L      1.3;
      BLD   103;
      A(    ;
      O     I    150.1;
      O     I      0.1;
      )     ;
      =     L      1.5;
      BLD   103;
      A     M      0.5;
      =     L      1.6;
      BLD   103;
      CALL #S704_LM_DC_OTR_CLAMP (
           Enable_Aux               := L      0.0,
           Adv_Amount               := 1,
           Ret_Amount               := 1,
           LS_Adv1                  := L      0.1,
           LS_Ret1                  := L      0.2,
           SOL_Adv                  := L      1.1,
           SOL_Ret                  := L      1.2,
           M_Ready                  := L      1.3,
           T_CHK1                   := T#4S,
           T_CHK2                   := T#4S,
           PB_Error_Rst             := L      1.5,
           M_FLICK                  := L      1.6,
           M_Adv_Err                := M   2152.6,
           M_Ret_Err                := M   2152.7,
           Visu_Adv                 := DB51.DBW  684,
           Visu_Ret                 := DB51.DBW  686);
      NOP   0;
NETWORK
TITLE =

      A     M   2002.7;
      =     L      0.0;
      BLD   103;
      A     I    268.0;
      =     L      0.1;
      BLD   103;
      A     I    268.1;
      =     L      0.2;
      BLD   103;
      A     Q    279.0;
      =     L      1.1;
      BLD   103;
      A     Q    279.1;
      =     L      1.2;
      BLD   103;
      AN    M   2004.0;
      AN    M   2004.1;
      AN    M   6060.1;
      AN    M   6460.0;
      AN    M   6480.0;
      AN    M   2004.2;
      A     M   2000.2;
      =     L      1.3;
      BLD   103;
      A(    ;
      O     I    150.1;
      O     I      0.1;
      )     ;
      =     L      1.5;
      BLD   103;
      A     M      0.5;
      =     L      1.6;
      BLD   103;
      CALL #S704_LM_DC_ASSY_CLAMP (
           Enable_Aux               := L      0.0,
           Adv_Amount               := 1,
           Ret_Amount               := 1,
           LS_Adv1                  := L      0.1,
           LS_Ret1                  := L      0.2,
           SOL_Adv                  := L      1.1,
           SOL_Ret                  := L      1.2,
           M_Ready                  := L      1.3,
           T_CHK1                   := T#4S,
           T_CHK2                   := T#4S,
           PB_Error_Rst             := L      1.5,
           M_FLICK                  := L      1.6,
           M_Adv_Err                := M   2153.0,
           M_Ret_Err                := M   2153.1,
           Visu_Adv                 := DB51.DBW  688,
           Visu_Ret                 := DB51.DBW  690);
      NOP   0;
NETWORK
TITLE =
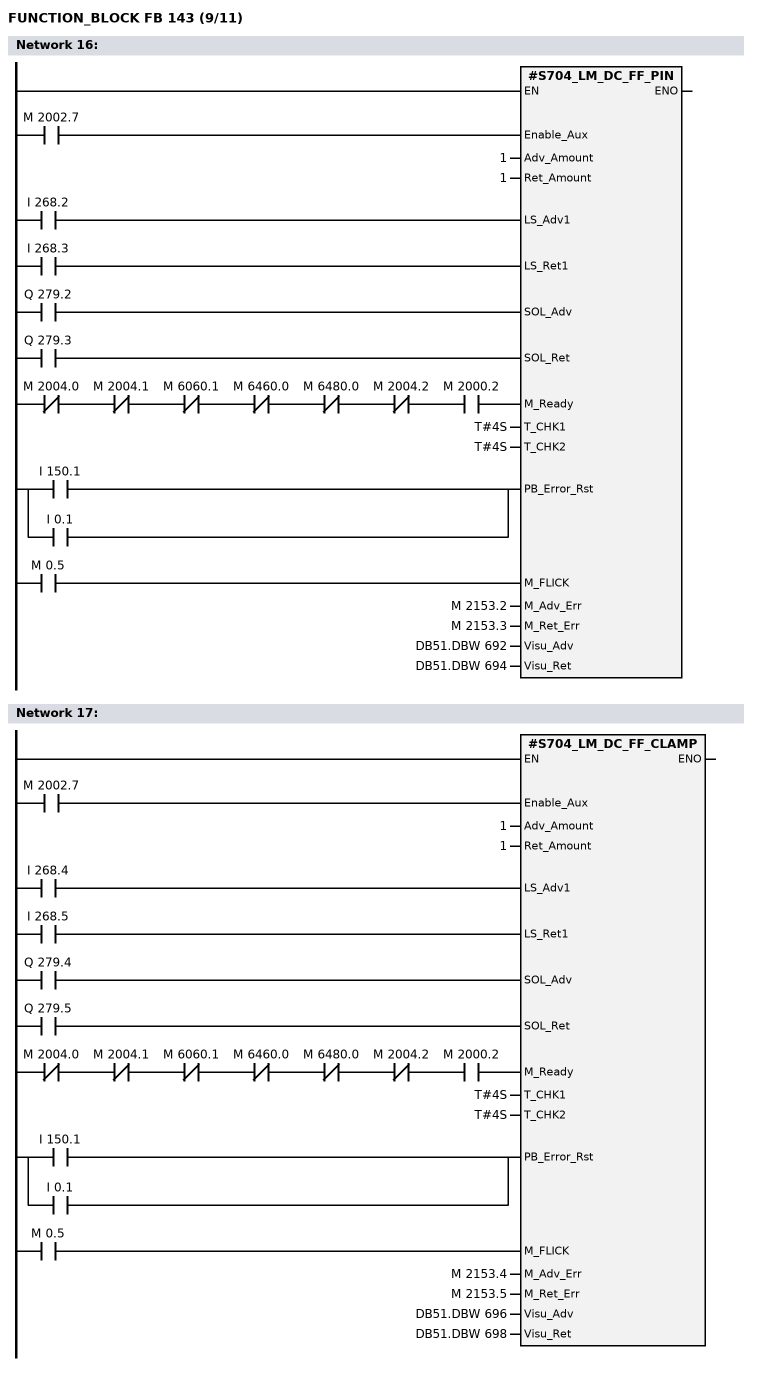

      A     M   2002.7;
      =     L      0.0;
      BLD   103;
      A     I    268.2;
      =     L      0.1;
      BLD   103;
      A     I    268.3;
      =     L      0.2;
      BLD   103;
      A     Q    279.2;
      =     L      1.1;
      BLD   103;
      A     Q    279.3;
      =     L      1.2;
      BLD   103;
      AN    M   2004.0;
      AN    M   2004.1;
      AN    M   6060.1;
      AN    M   6460.0;
      AN    M   6480.0;
      AN    M   2004.2;
      A     M   2000.2;
      =     L      1.3;
      BLD   103;
      A(    ;
      O     I    150.1;
      O     I      0.1;
      )     ;
      =     L      1.5;
      BLD   103;
      A     M      0.5;
      =     L      1.6;
      BLD   103;
      CALL #S704_LM_DC_FF_PIN (
           Enable_Aux               := L      0.0,
           Adv_Amount               := 1,
           Ret_Amount               := 1,
           LS_Adv1                  := L      0.1,
           LS_Ret1                  := L      0.2,
           SOL_Adv                  := L      1.1,
           SOL_Ret                  := L      1.2,
           M_Ready                  := L      1.3,
           T_CHK1                   := T#4S,
           T_CHK2                   := T#4S,
           PB_Error_Rst             := L      1.5,
           M_FLICK                  := L      1.6,
           M_Adv_Err                := M   2153.2,
           M_Ret_Err                := M   2153.3,
           Visu_Adv                 := DB51.DBW  692,
           Visu_Ret                 := DB51.DBW  694);
      NOP   0;
NETWORK
TITLE =

      A     M   2002.7;
      =     L      0.0;
      BLD   103;
      A     I    268.4;
      =     L      0.1;
      BLD   103;
      A     I    268.5;
      =     L      0.2;
      BLD   103;
      A     Q    279.4;
      =     L      1.1;
      BLD   103;
      A     Q    279.5;
      =     L      1.2;
      BLD   103;
      AN    M   2004.0;
      AN    M   2004.1;
      AN    M   6060.1;
      AN    M   6460.0;
      AN    M   6480.0;
      AN    M   2004.2;
      A     M   2000.2;
      =     L      1.3;
      BLD   103;
      A(    ;
      O     I    150.1;
      O     I      0.1;
      )     ;
      =     L      1.5;
      BLD   103;
      A     M      0.5;
      =     L      1.6;
      BLD   103;
      CALL #S704_LM_DC_FF_CLAMP (
           Enable_Aux               := L      0.0,
           Adv_Amount               := 1,
           Ret_Amount               := 1,
           LS_Adv1                  := L      0.1,
           LS_Ret1                  := L      0.2,
           SOL_Adv                  := L      1.1,
           SOL_Ret                  := L      1.2,
           M_Ready                  := L      1.3,
           T_CHK1                   := T#4S,
           T_CHK2                   := T#4S,
           PB_Error_Rst             := L      1.5,
           M_FLICK                  := L      1.6,
           M_Adv_Err                := M   2153.4,
           M_Ret_Err                := M   2153.5,
           Visu_Adv                 := DB51.DBW  696,
           Visu_Ret                 := DB51.DBW  698);
      NOP   0;
NETWORK
TITLE =
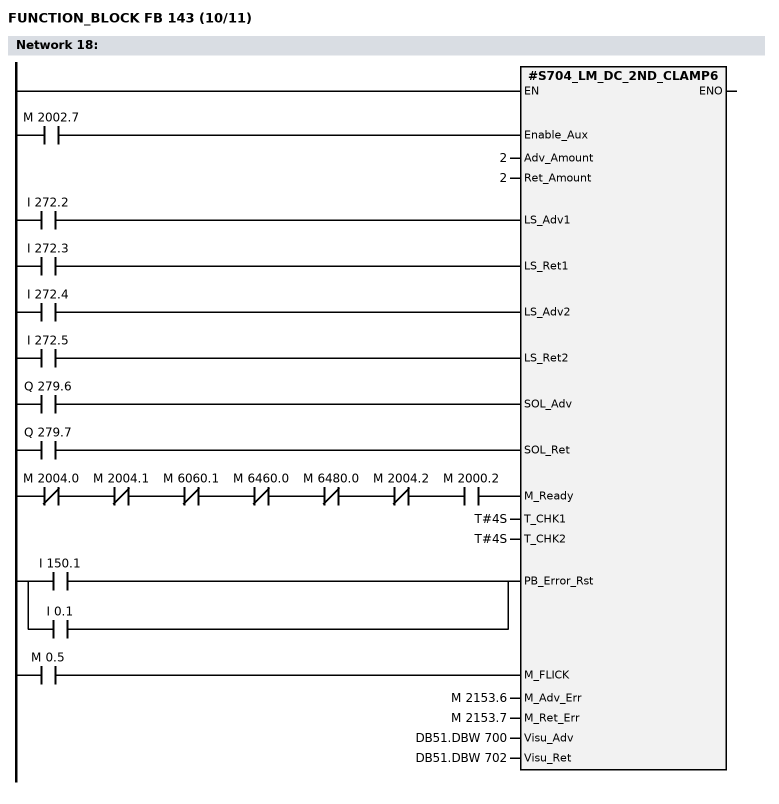

      A     M   2002.7;
      =     L      0.0;
      BLD   103;
      A     I    272.2;
      =     L      0.1;
      BLD   103;
      A     I    272.3;
      =     L      0.2;
      BLD   103;
      A     I    272.4;
      =     L      0.3;
      BLD   103;
      A     I    272.5;
      =     L      0.4;
      BLD   103;
      A     Q    279.6;
      =     L      1.1;
      BLD   103;
      A     Q    279.7;
      =     L      1.2;
      BLD   103;
      AN    M   2004.0;
      AN    M   2004.1;
      AN    M   6060.1;
      AN    M   6460.0;
      AN    M   6480.0;
      AN    M   2004.2;
      A     M   2000.2;
      =     L      1.3;
      BLD   103;
      A(    ;
      O     I    150.1;
      O     I      0.1;
      )     ;
      =     L      1.5;
      BLD   103;
      A     M      0.5;
      =     L      1.6;
      BLD   103;
      CALL #S704_LM_DC_2ND_CLAMP6 (
           Enable_Aux               := L      0.0,
           Adv_Amount               := 2,
           Ret_Amount               := 2,
           LS_Adv1                  := L      0.1,
           LS_Ret1                  := L      0.2,
           LS_Adv2                  := L      0.3,
           LS_Ret2                  := L      0.4,
           SOL_Adv                  := L      1.1,
           SOL_Ret                  := L      1.2,
           M_Ready                  := L      1.3,
           T_CHK1                   := T#4S,
           T_CHK2                   := T#4S,
           PB_Error_Rst             := L      1.5,
           M_FLICK                  := L      1.6,
           M_Adv_Err                := M   2153.6,
           M_Ret_Err                := M   2153.7,
           Visu_Adv                 := DB51.DBW  700,
           Visu_Ret                 := DB51.DBW  702);
      NOP   0;
NETWORK
TITLE =
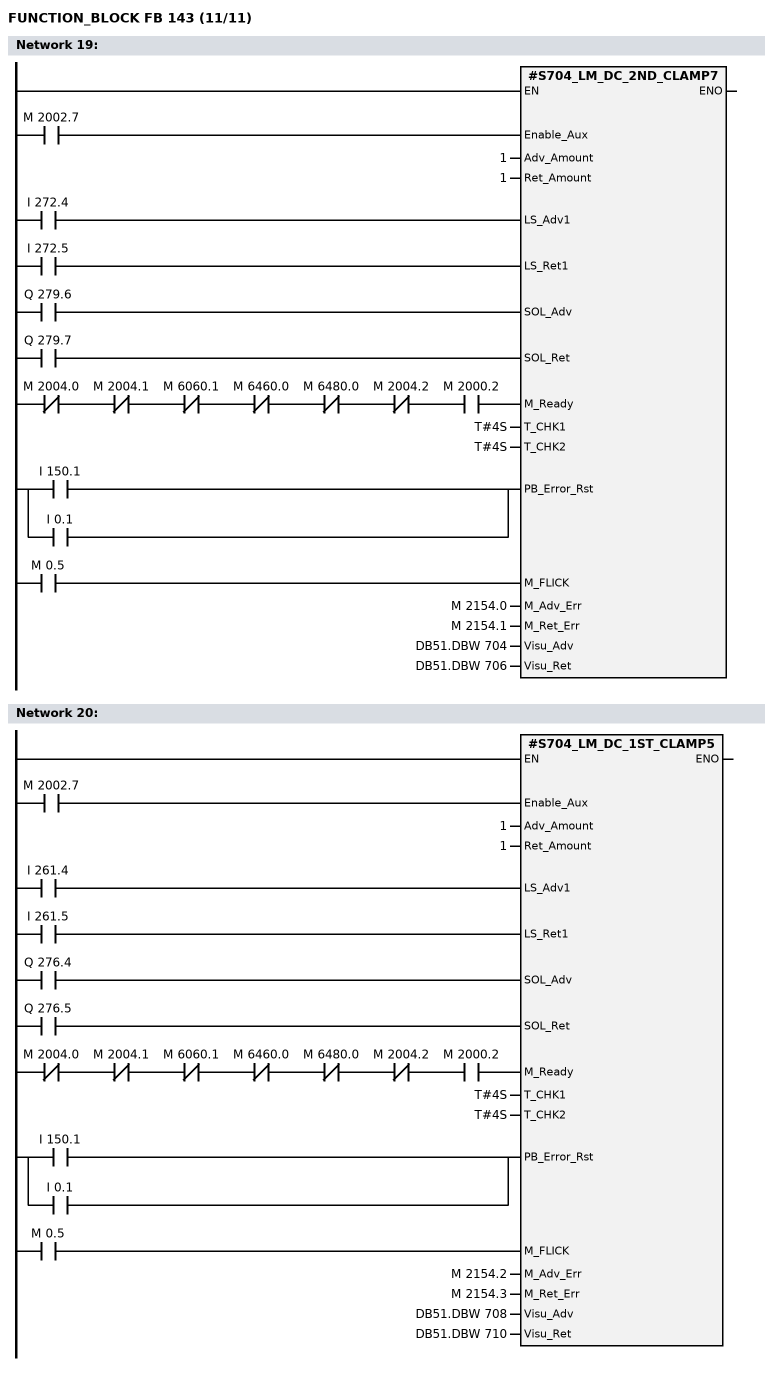

      A     M   2002.7;
      =     L      0.0;
      BLD   103;
      A     I    272.4;
      =     L      0.1;
      BLD   103;
      A     I    272.5;
      =     L      0.2;
      BLD   103;
      A     Q    279.6;
      =     L      1.1;
      BLD   103;
      A     Q    279.7;
      =     L      1.2;
      BLD   103;
      AN    M   2004.0;
      AN    M   2004.1;
      AN    M   6060.1;
      AN    M   6460.0;
      AN    M   6480.0;
      AN    M   2004.2;
      A     M   2000.2;
      =     L      1.3;
      BLD   103;
      A(    ;
      O     I    150.1;
      O     I      0.1;
      )     ;
      =     L      1.5;
      BLD   103;
      A     M      0.5;
      =     L      1.6;
      BLD   103;
      CALL #S704_LM_DC_2ND_CLAMP7 (
           Enable_Aux               := L      0.0,
           Adv_Amount               := 1,
           Ret_Amount               := 1,
           LS_Adv1                  := L      0.1,
           LS_Ret1                  := L      0.2,
           SOL_Adv                  := L      1.1,
           SOL_Ret                  := L      1.2,
           M_Ready                  := L      1.3,
           T_CHK1                   := T#4S,
           T_CHK2                   := T#4S,
           PB_Error_Rst             := L      1.5,
           M_FLICK                  := L      1.6,
           M_Adv_Err                := M   2154.0,
           M_Ret_Err                := M   2154.1,
           Visu_Adv                 := DB51.DBW  704,
           Visu_Ret                 := DB51.DBW  706);
      NOP   0;
NETWORK
TITLE =

      A     M   2002.7;
      =     L      0.0;
      BLD   103;
      A     I    261.4;
      =     L      0.1;
      BLD   103;
      A     I    261.5;
      =     L      0.2;
      BLD   103;
      A     Q    276.4;
      =     L      1.1;
      BLD   103;
      A     Q    276.5;
      =     L      1.2;
      BLD   103;
      AN    M   2004.0;
      AN    M   2004.1;
      AN    M   6060.1;
      AN    M   6460.0;
      AN    M   6480.0;
      AN    M   2004.2;
      A     M   2000.2;
      =     L      1.3;
      BLD   103;
      A(    ;
      O     I    150.1;
      O     I      0.1;
      )     ;
      =     L      1.5;
      BLD   103;
      A     M      0.5;
      =     L      1.6;
      BLD   103;
      CALL #S704_LM_DC_1ST_CLAMP5 (
           Enable_Aux               := L      0.0,
           Adv_Amount               := 1,
           Ret_Amount               := 1,
           LS_Adv1                  := L      0.1,
           LS_Ret1                  := L      0.2,
           SOL_Adv                  := L      1.1,
           SOL_Ret                  := L      1.2,
           M_Ready                  := L      1.3,
           T_CHK1                   := T#4S,
           T_CHK2                   := T#4S,
           PB_Error_Rst             := L      1.5,
           M_FLICK                  := L      1.6,
           M_Adv_Err                := M   2154.2,
           M_Ret_Err                := M   2154.3,
           Visu_Adv                 := DB51.DBW  708,
           Visu_Ret                 := DB51.DBW  710);
      NOP   0;
END_FUNCTION_BLOCK

DATA_BLOCK DB 143
TITLE =
VERSION : 0.0

